LIN {X 0,Y 188.988,Z 308.592,A -85,B 0,C 180,E1 -22467.201,E2 -22467.201} C_VEL
LIN {X 0,Y 185.39,Z 303.655,A -85,B 0,C 180,E1 -22469.376,E2 -22469.376} C_VEL
LIN {X 0,Y 183.716,Z 298.969,A -85,B 0,C 180,E1 -22473.901,E2 -22473.901} C_VEL
LIN {X 0,Y 182.459,Z 295.961,A -85,B 0,C 180,E1 -22477.581,E2 -22477.581} C_VEL
LIN {X 0,Y 181.404,Z 292.928,A -85,B 0,C 180,E1 -22481.945,E2 -22481.945} C_VEL
LIN {X 0,Y 180.335,Z 289.551,A -85,B 0,C 180,E1 -22488.764,E2 -22488.764} C_VEL
LIN {X 0,Y 179.767,Z 288.375,A -85,B 0,C 180,E1 -22493.265,E2 -22493.265} C_VEL
LIN {X 0,Y 179.829,Z 287.586,A -85,B 0,C 180,E1 -22500.001,E2 -22500.001} C_VEL
LIN {X 0,Y 180.049,Z 288.87,A -85,B 0,C 180,E1 -22507.094,E2 -22507.094} C_VEL
LIN {X 0,Y 180.404,Z 289.347,A -85,B 0,C 180,E1 -22508.966,E2 -22508.966} C_VEL
LIN {X 0,Y 181.337,Z 292.707,A -85,B 0,C 180,E1 -22515.742,E2 -22515.742} C_VEL
LIN {X 0,Y 182.454,Z 295.747,A -85,B 0,C 180,E1 -22520.285,E2 -22520.285} C_VEL
LIN {X 0,Y 183.828,Z 299.51,A -85,B 0,C 180,E1 -22524.87,E2 -22524.87} C_VEL
LIN {X 0,Y 185.464,Z 304.104,A -85,B 0,C 180,E1 -22529.514,E2 -22529.514} C_VEL
LIN {X 0,Y 186.625,Z 307.65,A -85,B 0,C 180,E1 -22532.354,E2 -22532.354} C_VEL
LIN {X 0,Y 190.377,Z 313.038,A -85,B 0,C 180,E1 -22534.503,E2 -22534.503} C_VEL
LIN {X 0,Y 194.923,Z 320.088,A -85,B 0,C 180,E1 -22536.853,E2 -22536.853} C_VEL
LIN {X 0,Y 200.843,Z 329.671,A -85,B 0,C 180,E1 -22539.608,E2 -22539.608} C_VEL
LIN {X 0,Y 207.054,Z 341.003,A -85,B 0,C 180,E1 -22542.242,E2 -22542.242} C_VEL
LIN {X 0,Y 213.308,Z 354.054,A -85,B 0,C 180,E1 -22544.675,E2 -22544.675} C_VEL
LIN {X 0,Y 215.63,Z 359.84,A -85,B 0,C 180,E1 -22545.558,E2 -22545.558} C_VEL
LIN {X 0,Y 216.978,Z 371.187,A -85,B 0,C 180,E1 -22546.403,E2 -22546.403} C_VEL
LIN {X 0,Y 213.581,Z 427.914,A -85,B 0,C 180,E1 -22548.075,E2 -22548.075} C_VEL
LIN {X 0,Y 211.9,Z 441.326,A -85,B 0,C 180,E1 -22548.763,E2 -22548.763} C_VEL
LIN {X 0,Y 209.528,Z 454.408,A -85,B 0,C 180,E1 -22549.784,E2 -22549.784} C_VEL
LIN {X 0,Y 206.842,Z 466.094,A -85,B 0,C 180,E1 -22551.055,E2 -22551.055} C_VEL
LIN {X 0,Y 203.672,Z 477.504,A -85,B 0,C 180,E1 -22552.686,E2 -22552.686} C_VEL
LIN {X 0,Y 200.113,Z 487.996,A -85,B 0,C 180,E1 -22554.586,E2 -22554.586} C_VEL
LIN {X 0,Y 196.107,Z 497.993,A -85,B 0,C 180,E1 -22556.872,E2 -22556.872} C_VEL
LIN {X 0,Y 192.484,Z 506.265,A -85,B 0,C 180,E1 -22559.259,E2 -22559.259} C_VEL
LIN {X 0,Y 188.562,Z 514.429,A -85,B 0,C 180,E1 -22562.232,E2 -22562.232} C_VEL
LIN {X 0,Y 185.25,Z 521.075,A -85,B 0,C 180,E1 -22565.335,E2 -22565.335} C_VEL
LIN {X 0,Y 182.489,Z 526.45,A -85,B 0,C 180,E1 -22568.54,E2 -22568.54} C_VEL
LIN {X 0,Y 180.226,Z 530.729,A -85,B 0,C 180,E1 -22571.823,E2 -22571.823} C_VEL
LIN {X 0,Y 178.925,Z 533.018,A -85,B 0,C 180,E1 -22574.041,E2 -22574.041} C_VEL
LIN {X 0,Y 177.241,Z 536.394,A -85,B 0,C 180,E1 -22578.565,E2 -22578.565} C_VEL
LIN {X 0,Y 176.7,Z 537.498,A -85,B 0,C 180,E1 -22580.846,E2 -22580.846} C_VEL
LIN {X 0,Y 176.115,Z 538.572,A -85,B 0,C 180,E1 -22585.422,E2 -22585.422} C_VEL
LIN {X 0,Y 176.114,Z 538.233,A -85,B 0,C 180,E1 -22590,E2 -22590} C_VEL
LIN {X 0,Y 176.586,Z 536.474,A -85,B 0,C 180,E1 -22594.565,E2 -22594.565} C_VEL
LIN {X 0,Y 177.693,Z 533.161,A -85,B 0,C 180,E1 -22599.102,E2 -22599.102} C_VEL
LIN {X 0,Y 179.055,Z 529.638,A -85,B 0,C 180,E1 -22602.467,E2 -22602.467} C_VEL
LIN {X 0,Y 180.92,Z 525.106,A -85,B 0,C 180,E1 -22605.778,E2 -22605.778} C_VEL
LIN {X 0,Y 183.79,Z 518.335,A -85,B 0,C 180,E1 -22609.547,E2 -22609.547} C_VEL
LIN {X 0,Y 186.845,Z 511.095,A -85,B 0,C 180,E1 -22612.677,E2 -22612.677} C_VEL
LIN {X 0,Y 190.293,Z 502.209,A -85,B 0,C 180,E1 -22615.718,E2 -22615.718} C_VEL
LIN {X 0,Y 193.973,Z 492.174,A -85,B 0,C 180,E1 -22618.394,E2 -22618.394} C_VEL
LIN {X 0,Y 197.187,Z 482.065,A -85,B 0,C 180,E1 -22620.522,E2 -22620.522} C_VEL
LIN {X 0,Y 200.625,Z 469.958,A -85,B 0,C 180,E1 -22622.485,E2 -22622.485} C_VEL
LIN {X 0,Y 203.442,Z 457.934,A -85,B 0,C 180,E1 -22623.971,E2 -22623.971} C_VEL
LIN {X 0,Y 205.741,Z 444.65,A -85,B 0,C 180,E1 -22625.199,E2 -22625.199} C_VEL
LIN {X 0,Y 207.478,Z 431.116,A -85,B 0,C 180,E1 -22626.008,E2 -22626.008} C_VEL
LIN {X 0,Y 208.695,Z 413.538,A -85,B 0,C 180,E1 -22626.617,E2 -22626.617} C_VEL
LIN {X 0,Y 211.032,Z 367.372,A -85,B 0,C 180,E1 -22628.031,E2 -22628.031} C_VEL
LIN {X 0,Y 209.082,Z 351.343,A -85,B 0,C 180,E1 -22629.173,E2 -22629.173} C_VEL
LIN {X 0,Y 202.802,Z 337.342,A -85,B 0,C 180,E1 -22631.415,E2 -22631.415} C_VEL
LIN {X 0,Y 197.38,Z 326.733,A -85,B 0,C 180,E1 -22633.468,E2 -22633.468} C_VEL
LIN {X 0,Y 191.774,Z 317.194,A -85,B 0,C 180,E1 -22635.727,E2 -22635.727} C_VEL
LIN {X 0,Y 188.452,Z 311.954,A -85,B 0,C 180,E1 -22637.158,E2 -22637.158} C_VEL
LIN {X 0,Y 185.851,Z 307.521,A -85,B 0,C 180,E1 -22638.52,E2 -22638.52} C_VEL
LIN {X 0,Y 184.237,Z 302.058,A -85,B 0,C 180,E1 -22642.385,E2 -22642.385} C_VEL
LIN {X 0,Y 182.761,Z 297.513,A -85,B 0,C 180,E1 -22646.11,E2 -22646.11} C_VEL
LIN {X 0,Y 180.979,Z 292.372,A -85,B 0,C 180,E1 -22650.959,E2 -22650.959} C_VEL
LIN {X 0,Y 179.769,Z 289.141,A -85,B 0,C 180,E1 -22654.529,E2 -22654.529} C_VEL
LIN {X 0,Y 178.544,Z 285.92,A -85,B 0,C 180,E1 -22658.949,E2 -22658.949} C_VEL
LIN {X 0,Y 178.648,Z 285.846,A -85,B 0,C 180,E1 -22661.655,E2 -22661.655} C_VEL
LIN {X 0,Y 178.655,Z 285.843,A -85,B 0,C 180,E1 -22666.347,E2 -22666.347} C_VEL
LIN {X 0,Y 178.912,Z 285.807,A -85,B 0,C 180,E1 -22670.959,E2 -22670.959} C_VEL
LIN {X 0,Y 178.864,Z 285.81,A -85,B 0,C 180,E1 -22675.492,E2 -22675.492} C_VEL
LIN {X 0,Y 179.367,Z 285.749,A -85,B 0,C 180,E1 -22679.999,E2 -22679.999} C_VEL
LIN {X 0,Y 178.869,Z 285.817,A -85,B 0,C 180,E1 -22684.506,E2 -22684.506} C_VEL
LIN {X 0,Y 178.935,Z 285.816,A -85,B 0,C 180,E1 -22689.038,E2 -22689.038} C_VEL
LIN {X 0,Y 178.657,Z 285.857,A -85,B 0,C 180,E1 -22693.652,E2 -22693.652} C_VEL
LIN {X 0,Y 178.623,Z 286.004,A -85,B 0,C 180,E1 -22699.327,E2 -22699.327} C_VEL
LIN {X 0,Y 179.991,Z 289.783,A -85,B 0,C 180,E1 -22704.203,E2 -22704.203} C_VEL
LIN {X 0,Y 181.21,Z 293.097,A -85,B 0,C 180,E1 -22707.736,E2 -22707.736} C_VEL
LIN {X 0,Y 183.125,Z 298.362,A -85,B 0,C 180,E1 -22712.499,E2 -22712.499} C_VEL
LIN {X 0,Y 184.812,Z 303.336,A -85,B 0,C 180,E1 -22716.197,E2 -22716.197} C_VEL
LIN {X 0,Y 189.323,Z 310.216,A -85,B 0,C 180,E1 -22718.361,E2 -22718.361} C_VEL
LIN {X 0,Y 194.564,Z 318.216,A -85,B 0,C 180,E1 -22720.555,E2 -22720.555} C_VEL
LIN {X 0,Y 201.427,Z 330.245,A -85,B 0,C 180,E1 -22723.214,E2 -22723.214} C_VEL
LIN {X 0,Y 207.772,Z 343.107,A -85,B 0,C 180,E1 -22725.515,E2 -22725.515} C_VEL
LIN {X 0,Y 212.209,Z 353.469,A -85,B 0,C 180,E1 -22727.065,E2 -22727.065} C_VEL
LIN {X 0,Y 208.951,Z 409.204,A -85,B 0,C 180,E1 -22728.827,E2 -22728.827} C_VEL
LIN {X 0,Y 208.047,Z 415.053,A -85,B 0,C 180,E1 -22728.881,E2 -22728.881} C_VEL
LIN {X 0,Y 202.147,Z 433.973,A -85,B 0,C 180,E1 -22728.563,E2 -22728.563} C_VEL
LIN {X 0,Y 201.311,Z 437.801,A -85,B 0,C 180,E1 -22728.678,E2 -22728.678} C_VEL
LIN {X 0,Y 201.054,Z 439.716,A -85,B 0,C 180,E1 -22728.791,E2 -22728.791} C_VEL
LIN {X 0,Y 198.753,Z 453.725,A -85,B 0,C 180,E1 -22729.811,E2 -22729.811} C_VEL
LIN {X 0,Y 196.069,Z 466.519,A -85,B 0,C 180,E1 -22731.151,E2 -22731.151} C_VEL
LIN {X 0,Y 192.593,Z 479.599,A -85,B 0,C 180,E1 -22732.98,E2 -22732.98} C_VEL
LIN {X 0,Y 188.999,Z 491.567,A -85,B 0,C 180,E1 -22735.187,E2 -22735.187} C_VEL
LIN {X 0,Y 185.68,Z 501.033,A -85,B 0,C 180,E1 -22737.361,E2 -22737.361} C_VEL
LIN {X 0,Y 181.482,Z 511.683,A -85,B 0,C 180,E1 -22740.413,E2 -22740.413} C_VEL
LIN {X 0,Y 178.053,Z 520.388,A -85,B 0,C 180,E1 -22743.638,E2 -22743.638} C_VEL
LIN {X 0,Y 174.916,Z 528.205,A -85,B 0,C 180,E1 -22747.332,E2 -22747.332} C_VEL
LIN {X 0,Y 172.603,Z 534.285,A -85,B 0,C 180,E1 -22750.99,E2 -22750.99} C_VEL
LIN {X 0,Y 170.858,Z 538.9,A -85,B 0,C 180,E1 -22754.493,E2 -22754.493} C_VEL
LIN {X 0,Y 169.722,Z 542.492,A -85,B 0,C 180,E1 -22758.051,E2 -22758.051} C_VEL
LIN {X 0,Y 169.28,Z 544.407,A -85,B 0,C 180,E1 -22760.441,E2 -22760.441} C_VEL
LIN {X 0,Y 168.849,Z 547.061,A -85,B 0,C 180,E1 -22765.225,E2 -22765.225} C_VEL
LIN {X 0,Y 168.983,Z 548.218,A -85,B 0,C 180,E1 -22770,E2 -22770} C_VEL
LIN {X 0,Y 168.89,Z 548.208,A -85,B 0,C 180,E1 -22772.921,E2 -22772.921} C_VEL
LIN {X 0,Y 168.991,Z 547.226,A -85,B 0,C 180,E1 -22777.167,E2 -22777.167} C_VEL
LIN {X 0,Y 169.78,Z 544.762,A -85,B 0,C 180,E1 -22781.945,E2 -22781.945} C_VEL
LIN {X 0,Y 170.968,Z 541.886,A -85,B 0,C 180,E1 -22785.497,E2 -22785.497} C_VEL
LIN {X 0,Y 173.498,Z 536.673,A -85,B 0,C 180,E1 -22790.14,E2 -22790.14} C_VEL
LIN {X 0,Y 175.919,Z 531.55,A -85,B 0,C 180,E1 -22793.547,E2 -22793.547} C_VEL
LIN {X 0,Y 179.575,Z 524.164,A -85,B 0,C 180,E1 -22797.378,E2 -22797.378} C_VEL
LIN {X 0,Y 183.322,Z 516.339,A -85,B 0,C 180,E1 -22800.528,E2 -22800.528} C_VEL
LIN {X 0,Y 187.683,Z 506.803,A -85,B 0,C 180,E1 -22803.526,E2 -22803.526} C_VEL
LIN {X 0,Y 191.637,Z 497.209,A -85,B 0,C 180,E1 -22805.928,E2 -22805.928} C_VEL
LIN {X 0,Y 195.407,Z 486.819,A -85,B 0,C 180,E1 -22808.018,E2 -22808.018} C_VEL
LIN {X 0,Y 199.458,Z 473.997,A -85,B 0,C 180,E1 -22810.019,E2 -22810.019} C_VEL
LIN {X 0,Y 202.815,Z 461.325,A -85,B 0,C 180,E1 -22811.507,E2 -22811.507} C_VEL
LIN {X 0,Y 205.587,Z 448.261,A -85,B 0,C 180,E1 -22812.632,E2 -22812.632} C_VEL
LIN {X 0,Y 207.681,Z 434.633,A -85,B 0,C 180,E1 -22813.435,E2 -22813.435} C_VEL
LIN {X 0,Y 209.176,Z 417.644,A -85,B 0,C 180,E1 -22814.044,E2 -22814.044} C_VEL
LIN {X 0,Y 212.691,Z 361.582,A -85,B 0,C 180,E1 -22815.805,E2 -22815.805} C_VEL
LIN {X 0,Y 206.911,Z 348.829,A -85,B 0,C 180,E1 -22818.115,E2 -22818.115} C_VEL
LIN {X 0,Y 201.177,Z 337.852,A -85,B 0,C 180,E1 -22820.553,E2 -22820.553} C_VEL
LIN {X 0,Y 195.155,Z 327.838,A -85,B 0,C 180,E1 -22823.331,E2 -22823.331} C_VEL
LIN {X 0,Y 189.772,Z 319.519,A -85,B 0,C 180,E1 -22826.095,E2 -22826.095} C_VEL
LIN {X 0,Y 186.099,Z 314.359,A -85,B 0,C 180,E1 -22828.162,E2 -22828.162} C_VEL
LIN {X 0,Y 181.851,Z 308.686,A -85,B 0,C 180,E1 -22830.802,E2 -22830.802} C_VEL
LIN {X 0,Y 178.233,Z 303.751,A -85,B 0,C 180,E1 -22833.509,E2 -22833.509} C_VEL
LIN {X 0,Y 176.472,Z 299.364,A -85,B 0,C 180,E1 -22838.997,E2 -22838.997} C_VEL
LIN {X 0,Y 175.428,Z 296.432,A -85,B 0,C 180,E1 -22843.715,E2 -22843.715} C_VEL
LIN {X 0,Y 174.827,Z 294.233,A -85,B 0,C 180,E1 -22848.405,E2 -22848.405} C_VEL
LIN {X 0,Y 174.62,Z 293.43,A -85,B 0,C 180,E1 -22850.736,E2 -22850.736} C_VEL
LIN {X 0,Y 174.209,Z 292.288,A -85,B 0,C 180,E1 -22857.689,E2 -22857.689} C_VEL
LIN {X 0,Y 174.368,Z 292.137,A -85,B 0,C 180,E1 -22860.001,E2 -22860.001} C_VEL
LIN {X 0,Y 174.572,Z 293.41,A -85,B 0,C 180,E1 -22867.151,E2 -22867.151} C_VEL
LIN {X 0,Y 174.898,Z 293.994,A -85,B 0,C 180,E1 -22869.25,E2 -22869.25} C_VEL
LIN {X 0,Y 175.921,Z 297.612,A -85,B 0,C 180,E1 -22876.508,E2 -22876.508} C_VEL
LIN {X 0,Y 176.956,Z 300.581,A -85,B 0,C 180,E1 -22880.944,E2 -22880.944} C_VEL
LIN {X 0,Y 178.332,Z 304.501,A -85,B 0,C 180,E1 -22885.691,E2 -22885.691} C_VEL
LIN {X 0,Y 179.408,Z 307.362,A -85,B 0,C 180,E1 -22888.426,E2 -22888.426} C_VEL
LIN {X 0,Y 183.53,Z 313.038,A -85,B 0,C 180,E1 -22891.21,E2 -22891.21} C_VEL
LIN {X 0,Y 188.311,Z 320.152,A -85,B 0,C 180,E1 -22894.044,E2 -22894.044} C_VEL
LIN {X 0,Y 191.838,Z 325.708,A -85,B 0,C 180,E1 -22895.943,E2 -22895.943} C_VEL
LIN {X 0,Y 197.44,Z 335.085,A -85,B 0,C 180,E1 -22898.694,E2 -22898.694} C_VEL
LIN {X 0,Y 203.749,Z 346.971,A -85,B 0,C 180,E1 -22901.501,E2 -22901.501} C_VEL
LIN {X 0,Y 209.488,Z 359.433,A -85,B 0,C 180,E1 -22903.85,E2 -22903.85} C_VEL
LIN {X 0,Y 210.867,Z 363.303,A -85,B 0,C 180,E1 -22904.421,E2 -22904.421} C_VEL
LIN {X 0,Y 211.836,Z 372.835,A -85,B 0,C 180,E1 -22905.125,E2 -22905.125} C_VEL
LIN {X 0,Y 208.375,Z 427.933,A -85,B 0,C 180,E1 -22906.767,E2 -22906.767} C_VEL
LIN {X 0,Y 206.627,Z 441.435,A -85,B 0,C 180,E1 -22907.468,E2 -22907.468} C_VEL
LIN {X 0,Y 204.15,Z 454.506,A -85,B 0,C 180,E1 -22908.495,E2 -22908.495} C_VEL
LIN {X 0,Y 201.385,Z 466.19,A -85,B 0,C 180,E1 -22909.789,E2 -22909.789} C_VEL
LIN {X 0,Y 198.045,Z 477.602,A -85,B 0,C 180,E1 -22911.435,E2 -22911.435} C_VEL
LIN {X 0,Y 194.365,Z 488.1,A -85,B 0,C 180,E1 -22913.372,E2 -22913.372} C_VEL
LIN {X 0,Y 190.195,Z 498.105,A -85,B 0,C 180,E1 -22915.702,E2 -22915.702} C_VEL
LIN {X 0,Y 186.413,Z 506.385,A -85,B 0,C 180,E1 -22918.142,E2 -22918.142} C_VEL
LIN {X 0,Y 182.303,Z 514.558,A -85,B 0,C 180,E1 -22921.192,E2 -22921.192} C_VEL
LIN {X 0,Y 178.787,Z 521.213,A -85,B 0,C 180,E1 -22924.38,E2 -22924.38} C_VEL
LIN {X 0,Y 175.863,Z 526.599,A -85,B 0,C 180,E1 -22927.689,E2 -22927.689} C_VEL
LIN {X 0,Y 173.47,Z 530.888,A -85,B 0,C 180,E1 -22931.088,E2 -22931.088} C_VEL
LIN {X 0,Y 172.075,Z 533.182,A -85,B 0,C 180,E1 -22933.388,E2 -22933.388} C_VEL
LIN {X 0,Y 170.27,Z 536.568,A -85,B 0,C 180,E1 -22938.09,E2 -22938.09} C_VEL
LIN {X 0,Y 169.674,Z 537.682,A -85,B 0,C 180,E1 -22940.463,E2 -22940.463} C_VEL
LIN {X 0,Y 169.028,Z 538.768,A -85,B 0,C 180,E1 -22945.23,E2 -22945.23} C_VEL
LIN {X 0,Y 169.024,Z 538.441,A -85,B 0,C 180,E1 -22950,E2 -22950} C_VEL
LIN {X 0,Y 169.52,Z 536.696,A -85,B 0,C 180,E1 -22954.756,E2 -22954.756} C_VEL
LIN {X 0,Y 170.691,Z 533.4,A -85,B 0,C 180,E1 -22959.479,E2 -22959.479} C_VEL
LIN {X 0,Y 172.727,Z 528.497,A -85,B 0,C 180,E1 -22964.13,E2 -22964.13} C_VEL
LIN {X 0,Y 174.915,Z 523.6,A -85,B 0,C 180,E1 -22967.538,E2 -22967.538} C_VEL
LIN {X 0,Y 178.166,Z 516.415,A -85,B 0,C 180,E1 -22971.4,E2 -22971.4} C_VEL
LIN {X 0,Y 181.505,Z 508.678,A -85,B 0,C 180,E1 -22974.597,E2 -22974.597} C_VEL
LIN {X 0,Y 185.368,Z 499.143,A -85,B 0,C 180,E1 -22977.674,E2 -22977.674} C_VEL
LIN {X 0,Y 188.94,Z 489.408,A -85,B 0,C 180,E1 -22980.142,E2 -22980.142} C_VEL
LIN {X 0,Y 192.342,Z 478.69,A -85,B 0,C 180,E1 -22982.301,E2 -22982.301} C_VEL
LIN {X 0,Y 195.657,Z 467.131,A -85,B 0,C 180,E1 -22984.071,E2 -22984.071} C_VEL
LIN {X 0,Y 198.523,Z 454.168,A -85,B 0,C 180,E1 -22985.583,E2 -22985.583} C_VEL
LIN {X 0,Y 200.692,Z 441.123,A -85,B 0,C 180,E1 -22986.683,E2 -22986.683} C_VEL
LIN {X 0,Y 202.257,Z 428.164,A -85,B 0,C 180,E1 -22987.39,E2 -22987.39} C_VEL
LIN {X 0,Y 205.638,Z 368.57,A -85,B 0,C 180,E1 -22989.267,E2 -22989.267} C_VEL
LIN {X 0,Y 203.986,Z 354.351,A -85,B 0,C 180,E1 -22990.318,E2 -22990.318} C_VEL
LIN {X 0,Y 198.265,Z 341.326,A -85,B 0,C 180,E1 -22992.492,E2 -22992.492} C_VEL
LIN {X 0,Y 193.104,Z 331.102,A -85,B 0,C 180,E1 -22994.565,E2 -22994.565} C_VEL
LIN {X 0,Y 187.912,Z 322.048,A -85,B 0,C 180,E1 -22996.788,E2 -22996.788} C_VEL
LIN {X 0,Y 184.709,Z 316.898,A -85,B 0,C 180,E1 -22998.25,E2 -22998.25} C_VEL
LIN {X 0,Y 181.35,Z 311.778,A -85,B 0,C 180,E1 -22999.876,E2 -22999.876} C_VEL
LIN {X 0,Y 178.713,Z 307.363,A -85,B 0,C 180,E1 -23001.418,E2 -23001.418} C_VEL
LIN {X 0,Y 177.335,Z 302.898,A -85,B 0,C 180,E1 -23004.924,E2 -23004.924} C_VEL
LIN {X 0,Y 175.96,Z 298.779,A -85,B 0,C 180,E1 -23008.718,E2 -23008.718} C_VEL
LIN {X 0,Y 174.787,Z 295.473,A -85,B 0,C 180,E1 -23012.2,E2 -23012.2} C_VEL
LIN {X 0,Y 172.929,Z 290.476,A -85,B 0,C 180,E1 -23018.544,E2 -23018.544} C_VEL
LIN {X 0,Y 171.589,Z 286.754,A -85,B 0,C 180,E1 -23025.47,E2 -23025.47} C_VEL
LIN {X 0,Y 171.848,Z 286.685,A -85,B 0,C 180,E1 -23030.584,E2 -23030.584} C_VEL
LIN {X 0,Y 171.813,Z 286.688,A -85,B 0,C 180,E1 -23035.307,E2 -23035.307} C_VEL
LIN {X 0,Y 172.329,Z 286.625,A -85,B 0,C 180,E1 -23039.999,E2 -23039.999} C_VEL
LIN {X 0,Y 171.818,Z 286.693,A -85,B 0,C 180,E1 -23044.692,E2 -23044.692} C_VEL
LIN {X 0,Y 171.87,Z 286.691,A -85,B 0,C 180,E1 -23049.413,E2 -23049.413} C_VEL
LIN {X 0,Y 171.647,Z 286.964,A -85,B 0,C 180,E1 -23053.315,E2 -23053.315} C_VEL
LIN {X 0,Y 172.896,Z 290.092,A -85,B 0,C 180,E1 -23058.976,E2 -23058.976} C_VEL
LIN {X 0,Y 174.536,Z 294.799,A -85,B 0,C 180,E1 -23065.011,E2 -23065.011} C_VEL
LIN {X 0,Y 176.266,Z 299.567,A -85,B 0,C 180,E1 -23069.893,E2 -23069.893} C_VEL
LIN {X 0,Y 177.686,Z 303.491,A -85,B 0,C 180,E1 -23073.206,E2 -23073.206} C_VEL
LIN {X 0,Y 181.057,Z 308.371,A -85,B 0,C 180,E1 -23075.097,E2 -23075.097} C_VEL
LIN {X 0,Y 185.961,Z 315.797,A -85,B 0,C 180,E1 -23077.474,E2 -23077.474} C_VEL
LIN {X 0,Y 190.798,Z 323.362,A -85,B 0,C 180,E1 -23079.609,E2 -23079.609} C_VEL
LIN {X 0,Y 197.137,Z 334.68,A -85,B 0,C 180,E1 -23082.204,E2 -23082.204} C_VEL
LIN {X 0,Y 203.357,Z 347.627,A -85,B 0,C 180,E1 -23084.598,E2 -23084.598} C_VEL
LIN {X 0,Y 206.717,Z 355.627,A -85,B 0,C 180,E1 -23085.844,E2 -23085.844} C_VEL
LIN {X 0,Y 202.135,Z 429.954,A -85,B 0,C 180,E1 -23088.276,E2 -23088.276} C_VEL
LIN {X 0,Y 201.054,Z 439.716,A -85,B 0,C 180,E1 -23088.791,E2 -23088.791} C_VEL
LIN {X 0,Y 199.788,Z 445.41,A -85,B 0,C 180,E1 -23089.055,E2 -23089.055} C_VEL
LIN {X 0,Y 195.958,Z 454.527,A -85,B 0,C 180,E1 -23089.273,E2 -23089.273} C_VEL
LIN {X 0,Y 191.716,Z 463.419,A -85,B 0,C 180,E1 -23089.648,E2 -23089.648} C_VEL
LIN {X 0,Y 189.822,Z 468.738,A -85,B 0,C 180,E1 -23090.164,E2 -23090.164} C_VEL
LIN {X 0,Y 186.5,Z 480.541,A -85,B 0,C 180,E1 -23091.899,E2 -23091.899} C_VEL
LIN {X 0,Y 183.013,Z 491.653,A -85,B 0,C 180,E1 -23094.021,E2 -23094.021} C_VEL
LIN {X 0,Y 178.929,Z 502.623,A -85,B 0,C 180,E1 -23096.641,E2 -23096.641} C_VEL
LIN {X 0,Y 175.293,Z 511.339,A -85,B 0,C 180,E1 -23099.258,E2 -23099.258} C_VEL
LIN {X 0,Y 171.658,Z 520.079,A -85,B 0,C 180,E1 -23102.575,E2 -23102.575} C_VEL
LIN {X 0,Y 168.197,Z 528.201,A -85,B 0,C 180,E1 -23106.549,E2 -23106.549} C_VEL
LIN {X 0,Y 165.857,Z 534.023,A -85,B 0,C 180,E1 -23110.185,E2 -23110.185} C_VEL
LIN {X 0,Y 163.985,Z 538.65,A -85,B 0,C 180,E1 -23113.825,E2 -23113.825} C_VEL
LIN {X 0,Y 162.739,Z 542.253,A -85,B 0,C 180,E1 -23117.53,E2 -23117.53} C_VEL
LIN {X 0,Y 161.904,Z 545.708,A -85,B 0,C 180,E1 -23122.518,E2 -23122.518} C_VEL
LIN {X 0,Y 161.755,Z 547.613,A -85,B 0,C 180,E1 -23127.51,E2 -23127.51} C_VEL
LIN {X 0,Y 161.894,Z 548.017,A -85,B 0,C 180,E1 -23130,E2 -23130} C_VEL
LIN {X 0,Y 161.795,Z 548.051,A -85,B 0,C 180,E1 -23132.49,E2 -23132.49} C_VEL
LIN {X 0,Y 161.928,Z 547.04,A -85,B 0,C 180,E1 -23137.482,E2 -23137.482} C_VEL
LIN {X 0,Y 162.791,Z 544.584,A -85,B 0,C 180,E1 -23142.466,E2 -23142.466} C_VEL
LIN {X 0,Y 164.096,Z 541.719,A -85,B 0,C 180,E1 -23146.164,E2 -23146.164} C_VEL
LIN {X 0,Y 166.807,Z 536.515,A -85,B 0,C 180,E1 -23150.985,E2 -23150.985} C_VEL
LIN {X 0,Y 169.371,Z 531.4,A -85,B 0,C 180,E1 -23154.516,E2 -23154.516} C_VEL
LIN {X 0,Y 173.246,Z 524.024,A -85,B 0,C 180,E1 -23158.467,E2 -23158.467} C_VEL
LIN {X 0,Y 177.196,Z 516.207,A -85,B 0,C 180,E1 -23161.703,E2 -23161.703} C_VEL
LIN {X 0,Y 181.793,Z 506.678,A -85,B 0,C 180,E1 -23164.765,E2 -23164.765} C_VEL
LIN {X 0,Y 186.336,Z 496.031,A -85,B 0,C 180,E1 -23167.452,E2 -23167.452} C_VEL
LIN {X 0,Y 190.287,Z 485.405,A -85,B 0,C 180,E1 -23169.576,E2 -23169.576} C_VEL
LIN {X 0,Y 194.072,Z 473.879,A -85,B 0,C 180,E1 -23171.367,E2 -23171.367} C_VEL
LIN {X 0,Y 197.564,Z 461.203,A -85,B 0,C 180,E1 -23172.869,E2 -23172.869} C_VEL
LIN {X 0,Y 200.551,Z 447.38,A -85,B 0,C 180,E1 -23174.058,E2 -23174.058} C_VEL
LIN {X 0,Y 202.742,Z 433.134,A -85,B 0,C 180,E1 -23174.873,E2 -23174.873} C_VEL
LIN {X 0,Y 204.401,Z 413.511,A -85,B 0,C 180,E1 -23175.547,E2 -23175.547} C_VEL
LIN {X 0,Y 207.608,Z 363.936,A -85,B 0,C 180,E1 -23177.128,E2 -23177.128} C_VEL
LIN {X 0,Y 201.268,Z 350.06,A -85,B 0,C 180,E1 -23179.842,E2 -23179.842} C_VEL
LIN {X 0,Y 195.295,Z 338.908,A -85,B 0,C 180,E1 -23182.602,E2 -23182.602} C_VEL
LIN {X 0,Y 189.819,Z 329.842,A -85,B 0,C 180,E1 -23185.383,E2 -23185.383} C_VEL
LIN {X 0,Y 185.485,Z 323.326,A -85,B 0,C 180,E1 -23187.808,E2 -23187.808} C_VEL
LIN {X 0,Y 183.331,Z 320.171,A -85,B 0,C 180,E1 -23189.115,E2 -23189.115} C_VEL
LIN {X 0,Y 179.443,Z 314.792,A -85,B 0,C 180,E1 -23191.667,E2 -23191.667} C_VEL
LIN {X 0,Y 175.385,Z 309.519,A -85,B 0,C 180,E1 -23194.68,E2 -23194.68} C_VEL
LIN {X 0,Y 171.063,Z 304.168,A -85,B 0,C 180,E1 -23198.616,E2 -23198.616} C_VEL
LIN {X 0,Y 170.003,Z 301.235,A -85,B 0,C 180,E1 -23203.18,E2 -23203.18} C_VEL
LIN {X 0,Y 169.334,Z 298.913,A -85,B 0,C 180,E1 -23208.024,E2 -23208.024} C_VEL
LIN {X 0,Y 169.15,Z 298.05,A -85,B 0,C 180,E1 -23210.434,E2 -23210.434} C_VEL
LIN {X 0,Y 168.67,Z 297.177,A -85,B 0,C 180,E1 -23215.221,E2 -23215.221} C_VEL
LIN {X 0,Y 168.906,Z 296.688,A -85,B 0,C 180,E1 -23220.001,E2 -23220.001} C_VEL
LIN {X 0,Y 169.114,Z 297.927,A -85,B 0,C 180,E1 -23227.189,E2 -23227.189} C_VEL
LIN {X 0,Y 169.406,Z 298.635,A -85,B 0,C 180,E1 -23229.553,E2 -23229.553} C_VEL
LIN {X 0,Y 169.909,Z 300.873,A -85,B 0,C 180,E1 -23234.371,E2 -23234.371} C_VEL
LIN {X 0,Y 170.867,Z 303.708,A -85,B 0,C 180,E1 -23239.212,E2 -23239.212} C_VEL
LIN {X 0,Y 172.147,Z 307.05,A -85,B 0,C 180,E1 -23243.457,E2 -23243.457} C_VEL
LIN {X 0,Y 176.113,Z 312.387,A -85,B 0,C 180,E1 -23246.837,E2 -23246.837} C_VEL
LIN {X 0,Y 178.142,Z 315.199,A -85,B 0,C 180,E1 -23248.355,E2 -23248.355} C_VEL
LIN {X 0,Y 181.763,Z 320.287,A -85,B 0,C 180,E1 -23250.82,E2 -23250.82} C_VEL
LIN {X 0,Y 185.491,Z 325.949,A -85,B 0,C 180,E1 -23253.12,E2 -23253.12} C_VEL
LIN {X 0,Y 189.11,Z 331.89,A -85,B 0,C 180,E1 -23255.173,E2 -23255.173} C_VEL
LIN {X 0,Y 194.164,Z 340.57,A -85,B 0,C 180,E1 -23257.781,E2 -23257.781} C_VEL
LIN {X 0,Y 199.896,Z 351.759,A -85,B 0,C 180,E1 -23260.475,E2 -23260.475} C_VEL
LIN {X 0,Y 205.015,Z 363.097,A -85,B 0,C 180,E1 -23262.699,E2 -23262.699} C_VEL
LIN {X 0,Y 206.108,Z 365.908,A -85,B 0,C 180,E1 -23263.166,E2 -23263.166} C_VEL
LIN {X 0,Y 206.863,Z 373.468,A -85,B 0,C 180,E1 -23263.753,E2 -23263.753} C_VEL
LIN {X 0,Y 203.268,Z 428.067,A -85,B 0,C 180,E1 -23265.398,E2 -23265.398} C_VEL
LIN {X 0,Y 201.469,Z 441.545,A -85,B 0,C 180,E1 -23266.108,E2 -23266.108} C_VEL
LIN {X 0,Y 198.903,Z 454.604,A -85,B 0,C 180,E1 -23267.143,E2 -23267.143} C_VEL
LIN {X 0,Y 196.02,Z 466.285,A -85,B 0,C 180,E1 -23268.449,E2 -23268.449} C_VEL
LIN {X 0,Y 192.279,Z 478.472,A -85,B 0,C 180,E1 -23270.245,E2 -23270.245} C_VEL
LIN {X 0,Y 188.258,Z 489.272,A -85,B 0,C 180,E1 -23272.317,E2 -23272.317} C_VEL
LIN {X 0,Y 183.501,Z 499.986,A -85,B 0,C 180,E1 -23274.937,E2 -23274.937} C_VEL
LIN {X 0,Y 178.934,Z 509.446,A -85,B 0,C 180,E1 -23277.979,E2 -23277.979} C_VEL
LIN {X 0,Y 174.771,Z 517.09,A -85,B 0,C 180,E1 -23281.148,E2 -23281.148} C_VEL
LIN {X 0,Y 171.209,Z 523.443,A -85,B 0,C 180,E1 -23284.569,E2 -23284.569} C_VEL
LIN {X 0,Y 168.404,Z 528.322,A -85,B 0,C 180,E1 -23287.939,E2 -23287.939} C_VEL
LIN {X 0,Y 165.962,Z 532.266,A -85,B 0,C 180,E1 -23291.482,E2 -23291.482} C_VEL
LIN {X 0,Y 164.182,Z 535.238,A -85,B 0,C 180,E1 -23295.118,E2 -23295.118} C_VEL
LIN {X 0,Y 162.67,Z 537.865,A -85,B 0,C 180,E1 -23300.048,E2 -23300.048} C_VEL
LIN {X 0,Y 161.946,Z 538.964,A -85,B 0,C 180,E1 -23305.021,E2 -23305.021} C_VEL
LIN {X 0,Y 161.935,Z 538.648,A -85,B 0,C 180,E1 -23310,E2 -23310} C_VEL
LIN {X 0,Y 162.447,Z 536.918,A -85,B 0,C 180,E1 -23314.964,E2 -23314.964} C_VEL
LIN {X 0,Y 163.708,Z 533.639,A -85,B 0,C 180,E1 -23319.888,E2 -23319.888} C_VEL
LIN {X 0,Y 165.237,Z 530.148,A -85,B 0,C 180,E1 -23323.528,E2 -23323.528} C_VEL
LIN {X 0,Y 167.322,Z 525.647,A -85,B 0,C 180,E1 -23327.098,E2 -23327.098} C_VEL
LIN {X 0,Y 170.508,Z 518.922,A -85,B 0,C 180,E1 -23331.14,E2 -23331.14} C_VEL
LIN {X 0,Y 173.85,Z 511.732,A -85,B 0,C 180,E1 -23334.479,E2 -23334.479} C_VEL
LIN {X 0,Y 177.637,Z 502.908,A -85,B 0,C 180,E1 -23337.701,E2 -23337.701} C_VEL
LIN {X 0,Y 181.658,Z 492.973,A -85,B 0,C 180,E1 -23340.515,E2 -23340.515} C_VEL
LIN {X 0,Y 185.147,Z 483.001,A -85,B 0,C 180,E1 -23342.745,E2 -23342.745} C_VEL
LIN {X 0,Y 188.728,Z 471.537,A -85,B 0,C 180,E1 -23344.717,E2 -23344.717} C_VEL
LIN {X 0,Y 191.7,Z 460.075,A -85,B 0,C 180,E1 -23346.238,E2 -23346.238} C_VEL
LIN {X 0,Y 194.162,Z 447.719,A -85,B 0,C 180,E1 -23347.484,E2 -23347.484} C_VEL
LIN {X 0,Y 196.24,Z 433.883,A -85,B 0,C 180,E1 -23348.435,E2 -23348.435} C_VEL
LIN {X 0,Y 197.456,Z 419.765,A -85,B 0,C 180,E1 -23349.012,E2 -23349.012} C_VEL
LIN {X 0,Y 200.365,Z 369.705,A -85,B 0,C 180,E1 -23350.567,E2 -23350.567} C_VEL
LIN {X 0,Y 198.883,Z 356.983,A -85,B 0,C 180,E1 -23351.565,E2 -23351.565} C_VEL
LIN {X 0,Y 192.971,Z 343.441,A -85,B 0,C 180,E1 -23353.972,E2 -23353.972} C_VEL
LIN {X 0,Y 187.433,Z 332.605,A -85,B 0,C 180,E1 -23356.372,E2 -23356.372} C_VEL
LIN {X 0,Y 181.632,Z 322.707,A -85,B 0,C 180,E1 -23359.097,E2 -23359.097} C_VEL
LIN {X 0,Y 178.164,Z 317.338,A -85,B 0,C 180,E1 -23360.864,E2 -23360.864} C_VEL
LIN {X 0,Y 174.821,Z 312.213,A -85,B 0,C 180,E1 -23362.705,E2 -23362.705} C_VEL
LIN {X 0,Y 171.559,Z 307.159,A -85,B 0,C 180,E1 -23364.824,E2 -23364.824} C_VEL
LIN {X 0,Y 170.08,Z 302.721,A -85,B 0,C 180,E1 -23368.9,E2 -23368.9} C_VEL
LIN {X 0,Y 168.866,Z 299.22,A -85,B 0,C 180,E1 -23372.753,E2 -23372.753} C_VEL
LIN {X 0,Y 167.442,Z 295.397,A -85,B 0,C 180,E1 -23377.804,E2 -23377.804} C_VEL
LIN {X 0,Y 166.287,Z 292.436,A -85,B 0,C 180,E1 -23382.791,E2 -23382.791} C_VEL
LIN {X 0,Y 165.962,Z 291.146,A -85,B 0,C 180,E1 -23385.28,E2 -23385.28} C_VEL
LIN {X 0,Y 165.274,Z 289.396,A -85,B 0,C 180,E1 -23390.206,E2 -23390.206} C_VEL
LIN {X 0,Y 164.923,Z 288.388,A -85,B 0,C 180,E1 -23395.11,E2 -23395.11} C_VEL
LIN {X 0,Y 165.325,Z 287.802,A -85,B 0,C 180,E1 -23399.999,E2 -23399.999} C_VEL
LIN {X 0,Y 165.022,Z 288.719,A -85,B 0,C 180,E1 -23404.885,E2 -23404.885} C_VEL
LIN {X 0,Y 165.565,Z 289.974,A -85,B 0,C 180,E1 -23409.775,E2 -23409.775} C_VEL
LIN {X 0,Y 166.079,Z 291.384,A -85,B 0,C 180,E1 -23413.276,E2 -23413.276} C_VEL
LIN {X 0,Y 167.362,Z 294.972,A -85,B 0,C 180,E1 -23419.629,E2 -23419.629} C_VEL
LIN {X 0,Y 168.741,Z 298.768,A -85,B 0,C 180,E1 -23424.613,E2 -23424.613} C_VEL
LIN {X 0,Y 170.318,Z 303.224,A -85,B 0,C 180,E1 -23429.331,E2 -23429.331} C_VEL
LIN {X 0,Y 171.217,Z 304.942,A -85,B 0,C 180,E1 -23430.272,E2 -23430.272} C_VEL
LIN {X 0,Y 175.383,Z 310.479,A -85,B 0,C 180,E1 -23432.749,E2 -23432.749} C_VEL
LIN {X 0,Y 179.262,Z 316.121,A -85,B 0,C 180,E1 -23434.849,E2 -23434.849} C_VEL
LIN {X 0,Y 182.774,Z 321.55,A -85,B 0,C 180,E1 -23436.614,E2 -23436.614} C_VEL
LIN {X 0,Y 187.362,Z 329.022,A -85,B 0,C 180,E1 -23438.751,E2 -23438.751} C_VEL
LIN {X 0,Y 193.082,Z 339.482,A -85,B 0,C 180,E1 -23441.225,E2 -23441.225} C_VEL
LIN {X 0,Y 198.88,Z 351.822,A -85,B 0,C 180,E1 -23443.59,E2 -23443.59} C_VEL
LIN {X 0,Y 201.328,Z 357.785,A -85,B 0,C 180,E1 -23444.559,E2 -23444.559} C_VEL
LIN {X 0,Y 196.654,Z 430.659,A -85,B 0,C 180,E1 -23446.998,E2 -23446.998} C_VEL
LIN {X 0,Y 194.869,Z 444.575,A -85,B 0,C 180,E1 -23447.802,E2 -23447.802} C_VEL
LIN {X 0,Y 192.404,Z 457.613,A -85,B 0,C 180,E1 -23448.892,E2 -23448.892} C_VEL
LIN {X 0,Y 189.822,Z 468.738,A -85,B 0,C 180,E1 -23450.164,E2 -23450.164} C_VEL
LIN {X 0,Y 187.879,Z 474.002,A -85,B 0,C 180,E1 -23450.755,E2 -23450.755} C_VEL
LIN {X 0,Y 183.175,Z 482.297,A -85,B 0,C 180,E1 -23451.565,E2 -23451.565} C_VEL
LIN {X 0,Y 178.206,Z 490.252,A -85,B 0,C 180,E1 -23452.573,E2 -23452.573} C_VEL
LIN {X 0,Y 175.885,Z 494.903,A -85,B 0,C 180,E1 -23453.48,E2 -23453.48} C_VEL
LIN {X 0,Y 171.433,Z 505.911,A -85,B 0,C 180,E1 -23456.397,E2 -23456.397} C_VEL
LIN {X 0,Y 167.221,Z 515.599,A -85,B 0,C 180,E1 -23459.713,E2 -23459.713} C_VEL
LIN {X 0,Y 163.613,Z 523.544,A -85,B 0,C 180,E1 -23463.191,E2 -23463.191} C_VEL
LIN {X 0,Y 160.695,Z 530.075,A -85,B 0,C 180,E1 -23466.821,E2 -23466.821} C_VEL
LIN {X 0,Y 158.428,Z 535.409,A -85,B 0,C 180,E1 -23470.567,E2 -23470.567} C_VEL
LIN {X 0,Y 156.555,Z 539.686,A -85,B 0,C 180,E1 -23474.375,E2 -23474.375} C_VEL
LIN {X 0,Y 155.203,Z 543.943,A -85,B 0,C 180,E1 -23479.565,E2 -23479.565} C_VEL
LIN {X 0,Y 154.842,Z 545.485,A -85,B 0,C 180,E1 -23482.174,E2 -23482.174} C_VEL
LIN {X 0,Y 154.678,Z 546.635,A -85,B 0,C 180,E1 -23484.786,E2 -23484.786} C_VEL
LIN {X 0,Y 154.792,Z 547.815,A -85,B 0,C 180,E1 -23490,E2 -23490} C_VEL
LIN {X 0,Y 154.696,Z 547.854,A -85,B 0,C 180,E1 -23492.604,E2 -23492.604} C_VEL
LIN {X 0,Y 154.861,Z 546.853,A -85,B 0,C 180,E1 -23497.825,E2 -23497.825} C_VEL
LIN {X 0,Y 155.826,Z 544.408,A -85,B 0,C 180,E1 -23503.033,E2 -23503.033} C_VEL
LIN {X 0,Y 157.251,Z 541.551,A -85,B 0,C 180,E1 -23506.888,E2 -23506.888} C_VEL
LIN {X 0,Y 160.151,Z 536.357,A -85,B 0,C 180,E1 -23511.901,E2 -23511.901} C_VEL
LIN {X 0,Y 162.885,Z 531.251,A -85,B 0,C 180,E1 -23515.56,E2 -23515.56} C_VEL
LIN {X 0,Y 166.991,Z 523.884,A -85,B 0,C 180,E1 -23519.637,E2 -23519.637} C_VEL
LIN {X 0,Y 171.165,Z 516.075,A -85,B 0,C 180,E1 -23522.959,E2 -23522.959} C_VEL
LIN {X 0,Y 175.99,Z 506.554,A -85,B 0,C 180,E1 -23526.087,E2 -23526.087} C_VEL
LIN {X 0,Y 180.281,Z 496.969,A -85,B 0,C 180,E1 -23528.589,E2 -23528.589} C_VEL
LIN {X 0,Y 184.861,Z 485.289,A -85,B 0,C 180,E1 -23530.98,E2 -23530.98} C_VEL
LIN {X 0,Y 188.793,Z 473.762,A -85,B 0,C 180,E1 -23532.794,E2 -23532.794} C_VEL
LIN {X 0,Y 192.429,Z 461.081,A -85,B 0,C 180,E1 -23534.305,E2 -23534.305} C_VEL
LIN {X 0,Y 195.392,Z 447.977,A -85,B 0,C 180,E1 -23535.448,E2 -23535.448} C_VEL
LIN {X 0,Y 197.669,Z 433.725,A -85,B 0,C 180,E1 -23536.291,E2 -23536.291} C_VEL
LIN {X 0,Y 199.303,Z 415.827,A -85,B 0,C 180,E1 -23536.921,E2 -23536.921} C_VEL
LIN {X 0,Y 202.687,Z 366.534,A -85,B 0,C 180,E1 -23538.489,E2 -23538.489} C_VEL
LIN {X 0,Y 197.073,Z 354.065,A -85,B 0,C 180,E1 -23541.055,E2 -23541.055} C_VEL
LIN {X 0,Y 191.734,Z 343.87,A -85,B 0,C 180,E1 -23543.68,E2 -23543.68} C_VEL
LIN {X 0,Y 186.228,Z 334.646,A -85,B 0,C 180,E1 -23546.653,E2 -23546.653} C_VEL
LIN {X 0,Y 182.755,Z 329.204,A -85,B 0,C 180,E1 -23548.725,E2 -23548.725} C_VEL
LIN {X 0,Y 180.38,Z 325.652,A -85,B 0,C 180,E1 -23550.25,E2 -23550.25} C_VEL
LIN {X 0,Y 177.112,Z 320.944,A -85,B 0,C 180,E1 -23552.53,E2 -23552.53} C_VEL
LIN {X 0,Y 173.207,Z 315.742,A -85,B 0,C 180,E1 -23555.59,E2 -23555.59} C_VEL
LIN {X 0,Y 168.613,Z 310.135,A -85,B 0,C 180,E1 -23559.888,E2 -23559.888} C_VEL
LIN {X 0,Y 164.15,Z 304.568,A -85,B 0,C 180,E1 -23565.749,E2 -23565.749} C_VEL
LIN {X 0,Y 163.692,Z 302.716,A -85,B 0,C 180,E1 -23570.112,E2 -23570.112} C_VEL
LIN {X 0,Y 163.461,Z 302.084,A -85,B 0,C 180,E1 -23572.59,E2 -23572.59} C_VEL
LIN {X 0,Y 163.445,Z 301.24,A -85,B 0,C 180,E1 -23580.001,E2 -23580.001} C_VEL
LIN {X 0,Y 163.646,Z 302.509,A -85,B 0,C 180,E1 -23587.403,E2 -23587.403} C_VEL
LIN {X 0,Y 163.889,Z 303.271,A -85,B 0,C 180,E1 -23589.878,E2 -23589.878} C_VEL
LIN {X 0,Y 164.707,Z 306.328,A -85,B 0,C 180,E1 -23596.103,E2 -23596.103} C_VEL
LIN {X 0,Y 170.478,Z 313.877,A -85,B 0,C 180,E1 -23602.897,E2 -23602.897} C_VEL
LIN {X 0,Y 175.413,Z 320.633,A -85,B 0,C 180,E1 -23607.114,E2 -23607.114} C_VEL
LIN {X 0,Y 179.275,Z 326.338,A -85,B 0,C 180,E1 -23609.921,E2 -23609.921} C_VEL
LIN {X 0,Y 182.866,Z 331.999,A -85,B 0,C 180,E1 -23612.26,E2 -23612.26} C_VEL
LIN {X 0,Y 187.864,Z 340.469,A -85,B 0,C 180,E1 -23615.186,E2 -23615.186} C_VEL
LIN {X 0,Y 192.818,Z 349.742,A -85,B 0,C 180,E1 -23617.799,E2 -23617.799} C_VEL
LIN {X 0,Y 197.641,Z 359.857,A -85,B 0,C 180,E1 -23620.13,E2 -23620.13} C_VEL
LIN {X 0,Y 201.421,Z 368.833,A -85,B 0,C 180,E1 -23621.861,E2 -23621.861} C_VEL
LIN {X 0,Y 201.915,Z 375.314,A -85,B 0,C 180,E1 -23622.347,E2 -23622.347} C_VEL
LIN {X 0,Y 198.273,Z 428.322,A -85,B 0,C 180,E1 -23623.965,E2 -23623.965} C_VEL
LIN {X 0,Y 196.432,Z 441.653,A -85,B 0,C 180,E1 -23624.677,E2 -23624.677} C_VEL
LIN {X 0,Y 193.769,Z 454.701,A -85,B 0,C 180,E1 -23625.718,E2 -23625.718} C_VEL
LIN {X 0,Y 190.762,Z 466.38,A -85,B 0,C 180,E1 -23627.034,E2 -23627.034} C_VEL
LIN {X 0,Y 186.882,Z 478.531,A -85,B 0,C 180,E1 -23628.843,E2 -23628.843} C_VEL
LIN {X 0,Y 182.688,Z 489.377,A -85,B 0,C 180,E1 -23630.955,E2 -23630.955} C_VEL
LIN {X 0,Y 177.74,Z 500.098,A -85,B 0,C 180,E1 -23633.622,E2 -23633.622} C_VEL
LIN {X 0,Y 172.944,Z 509.567,A -85,B 0,C 180,E1 -23636.729,E2 -23636.729} C_VEL
LIN {X 0,Y 168.558,Z 517.223,A -85,B 0,C 180,E1 -23639.978,E2 -23639.978} C_VEL
LIN {X 0,Y 164.52,Z 524.007,A -85,B 0,C 180,E1 -23643.779,E2 -23643.779} C_VEL
LIN {X 0,Y 160.921,Z 529.878,A -85,B 0,C 180,E1 -23648.209,E2 -23648.209} C_VEL
LIN {X 0,Y 158.457,Z 533.51,A -85,B 0,C 180,E1 -23651.913,E2 -23651.913} C_VEL
LIN {X 0,Y 156.361,Z 536.918,A -85,B 0,C 180,E1 -23657.013,E2 -23657.013} C_VEL
LIN {X 0,Y 155.66,Z 538.048,A -85,B 0,C 180,E1 -23659.595,E2 -23659.595} C_VEL
LIN {X 0,Y 154.865,Z 539.161,A -85,B 0,C 180,E1 -23664.792,E2 -23664.792} C_VEL
LIN {X 0,Y 154.835,Z 538.856,A -85,B 0,C 180,E1 -23670,E2 -23670} C_VEL
LIN {X 0,Y 155.385,Z 537.138,A -85,B 0,C 180,E1 -23675.19,E2 -23675.19} C_VEL
LIN {X 0,Y 156.737,Z 533.878,A -85,B 0,C 180,E1 -23680.332,E2 -23680.332} C_VEL
LIN {X 0,Y 158.995,Z 529.007,A -85,B 0,C 180,E1 -23685.379,E2 -23685.379} C_VEL
LIN {X 0,Y 161.442,Z 524.144,A -85,B 0,C 180,E1 -23689.056,E2 -23689.056} C_VEL
LIN {X 0,Y 165.057,Z 517.011,A -85,B 0,C 180,E1 -23693.194,E2 -23693.194} C_VEL
LIN {X 0,Y 168.728,Z 509.344,A -85,B 0,C 180,E1 -23696.6,E2 -23696.6} C_VEL
LIN {X 0,Y 172.926,Z 499.879,A -85,B 0,C 180,E1 -23699.858,E2 -23699.858} C_VEL
LIN {X 0,Y 176.862,Z 490.23,A -85,B 0,C 180,E1 -23702.442,E2 -23702.442} C_VEL
LIN {X 0,Y 180.551,Z 479.63,A -85,B 0,C 180,E1 -23704.699,E2 -23704.699} C_VEL
LIN {X 0,Y 184.168,Z 468.136,A -85,B 0,C 180,E1 -23706.555,E2 -23706.555} C_VEL
LIN {X 0,Y 187.269,Z 455.432,A -85,B 0,C 180,E1 -23708.122,E2 -23708.122} C_VEL
LIN {X 0,Y 189.791,Z 441.645,A -85,B 0,C 180,E1 -23709.34,E2 -23709.34} C_VEL
LIN {X 0,Y 191.591,Z 427.748,A -85,B 0,C 180,E1 -23710.12,E2 -23710.12} C_VEL
LIN {X 0,Y 195.156,Z 370.647,A -85,B 0,C 180,E1 -23711.959,E2 -23711.959} C_VEL
LIN {X 0,Y 194.011,Z 360.114,A -85,B 0,C 180,E1 -23712.813,E2 -23712.813} C_VEL
LIN {X 0,Y 188.851,Z 347.984,A -85,B 0,C 180,E1 -23715.056,E2 -23715.056} C_VEL
LIN {X 0,Y 183.758,Z 337.672,A -85,B 0,C 180,E1 -23717.404,E2 -23717.404} C_VEL
LIN {X 0,Y 177.996,Z 327.655,A -85,B 0,C 180,E1 -23720.279,E2 -23720.279} C_VEL
LIN {X 0,Y 174.73,Z 322.424,A -85,B 0,C 180,E1 -23722.057,E2 -23722.057} C_VEL
LIN {X 0,Y 171.88,Z 317.921,A -85,B 0,C 180,E1 -23723.727,E2 -23723.727} C_VEL
LIN {X 0,Y 167.926,Z 312.19,A -85,B 0,C 180,E1 -23726.237,E2 -23726.237} C_VEL
LIN {X 0,Y 164.351,Z 306.969,A -85,B 0,C 180,E1 -23728.949,E2 -23728.949} C_VEL
LIN {X 0,Y 163.033,Z 303.168,A -85,B 0,C 180,E1 -23733.086,E2 -23733.086} C_VEL
LIN {X 0,Y 161.961,Z 300.3,A -85,B 0,C 180,E1 -23737.011,E2 -23737.011} C_VEL
LIN {X 0,Y 160.851,Z 297.184,A -85,B 0,C 180,E1 -23742.19,E2 -23742.19} C_VEL
LIN {X 0,Y 160.461,Z 295.891,A -85,B 0,C 180,E1 -23744.763,E2 -23744.763} C_VEL
LIN {X 0,Y 159.794,Z 294.032,A -85,B 0,C 180,E1 -23749.867,E2 -23749.867} C_VEL
LIN {X 0,Y 159.473,Z 292.947,A -85,B 0,C 180,E1 -23754.942,E2 -23754.942} C_VEL
LIN {X 0,Y 159.84,Z 292.331,A -85,B 0,C 180,E1 -23759.999,E2 -23759.999} C_VEL
LIN {X 0,Y 159.794,Z 293.842,A -85,B 0,C 180,E1 -23767.581,E2 -23767.581} C_VEL
LIN {X 0,Y 160.465,Z 295.561,A -85,B 0,C 180,E1 -23772.649,E2 -23772.649} C_VEL
LIN {X 0,Y 161.274,Z 298.264,A -85,B 0,C 180,E1 -23777.76,E2 -23777.76} C_VEL
LIN {X 0,Y 162.603,Z 301.708,A -85,B 0,C 180,E1 -23782.891,E2 -23782.891} C_VEL
LIN {X 0,Y 163.564,Z 304.102,A -85,B 0,C 180,E1 -23785.617,E2 -23785.617} C_VEL
LIN {X 0,Y 167.655,Z 309.554,A -85,B 0,C 180,E1 -23788.712,E2 -23788.712} C_VEL
LIN {X 0,Y 172.524,Z 316.349,A -85,B 0,C 180,E1 -23791.804,E2 -23791.804} C_VEL
LIN {X 0,Y 176.029,Z 321.568,A -85,B 0,C 180,E1 -23793.81,E2 -23793.81} C_VEL
LIN {X 0,Y 181.53,Z 330.345,A -85,B 0,C 180,E1 -23796.673,E2 -23796.673} C_VEL
LIN {X 0,Y 187.629,Z 341.404,A -85,B 0,C 180,E1 -23799.55,E2 -23799.55} C_VEL
LIN {X 0,Y 193.319,Z 353.269,A -85,B 0,C 180,E1 -23802.044,E2 -23802.044} C_VEL
LIN {X 0,Y 196.064,Z 359.975,A -85,B 0,C 180,E1 -23803.211,E2 -23803.211} C_VEL
LIN {X 0,Y 191.383,Z 430.31,A -85,B 0,C 180,E1 -23805.593,E2 -23805.593} C_VEL
LIN {X 0,Y 189.522,Z 444.388,A -85,B 0,C 180,E1 -23806.41,E2 -23806.41} C_VEL
LIN {X 0,Y 186.848,Z 458.024,A -85,B 0,C 180,E1 -23807.571,E2 -23807.571} C_VEL
LIN {X 0,Y 183.725,Z 470.672,A -85,B 0,C 180,E1 -23809.075,E2 -23809.075} C_VEL
LIN {X 0,Y 180.061,Z 482.905,A -85,B 0,C 180,E1 -23810.997,E2 -23810.997} C_VEL
LIN {X 0,Y 176.258,Z 493.985,A -85,B 0,C 180,E1 -23813.267,E2 -23813.267} C_VEL
LIN {X 0,Y 175.885,Z 494.903,A -85,B 0,C 180,E1 -23813.48,E2 -23813.48} C_VEL
LIN {X 0,Y 173.498,Z 499.454,A -85,B 0,C 180,E1 -23814.462,E2 -23814.462} C_VEL
LIN {X 0,Y 168.112,Z 506.495,A -85,B 0,C 180,E1 -23815.94,E2 -23815.94} C_VEL
LIN {X 0,Y 162.704,Z 513.082,A -85,B 0,C 180,E1 -23817.678,E2 -23817.678} C_VEL
LIN {X 0,Y 160.34,Z 516.816,A -85,B 0,C 180,E1 -23819.061,E2 -23819.061} C_VEL
LIN {X 0,Y 156.128,Z 525.545,A -85,B 0,C 180,E1 -23823.248,E2 -23823.248} C_VEL
LIN {X 0,Y 153.296,Z 531.689,A -85,B 0,C 180,E1 -23827.065,E2 -23827.065} C_VEL
LIN {X 0,Y 150.991,Z 536.693,A -85,B 0,C 180,E1 -23830.985,E2 -23830.985} C_VEL
LIN {X 0,Y 149.196,Z 540.684,A -85,B 0,C 180,E1 -23834.985,E2 -23834.985} C_VEL
LIN {X 0,Y 148.2,Z 543.712,A -85,B 0,C 180,E1 -23839.066,E2 -23839.066} C_VEL
LIN {X 0,Y 147.605,Z 546.421,A -85,B 0,C 180,E1 -23844.536,E2 -23844.536} C_VEL
LIN {X 0,Y 147.715,Z 547.615,A -85,B 0,C 180,E1 -23850,E2 -23850} C_VEL
LIN {X 0,Y 147.607,Z 547.658,A -85,B 0,C 180,E1 -23852.729,E2 -23852.729} C_VEL
LIN {X 0,Y 147.624,Z 547.342,A -85,B 0,C 180,E1 -23855.464,E2 -23855.464} C_VEL
LIN {X 0,Y 148.224,Z 545.632,A -85,B 0,C 180,E1 -23860.933,E2 -23860.933} C_VEL
LIN {X 0,Y 149.79,Z 542.455,A -85,B 0,C 180,E1 -23866.35,E2 -23866.35} C_VEL
LIN {X 0,Y 151.852,Z 539,A -85,B 0,C 180,E1 -23870.311,E2 -23870.311} C_VEL
LIN {X 0,Y 154.89,Z 533.752,A -85,B 0,C 180,E1 -23874.842,E2 -23874.842} C_VEL
LIN {X 0,Y 158.838,Z 527.117,A -85,B 0,C 180,E1 -23879.124,E2 -23879.124} C_VEL
LIN {X 0,Y 163.693,Z 518.684,A -85,B 0,C 180,E1 -23883.189,E2 -23883.189} C_VEL
LIN {X 0,Y 168.556,Z 509.792,A -85,B 0,C 180,E1 -23886.452,E2 -23886.452} C_VEL
LIN {X 0,Y 172.956,Z 500.881,A -85,B 0,C 180,E1 -23889.037,E2 -23889.037} C_VEL
LIN {X 0,Y 177.465,Z 490.375,A -85,B 0,C 180,E1 -23891.478,E2 -23891.478} C_VEL
LIN {X 0,Y 182.092,Z 478.285,A -85,B 0,C 180,E1 -23893.621,E2 -23893.621} C_VEL
LIN {X 0,Y 185.805,Z 466.81,A -85,B 0,C 180,E1 -23895.17,E2 -23895.17} C_VEL
LIN {X 0,Y 189.087,Z 454.313,A -85,B 0,C 180,E1 -23896.449,E2 -23896.449} C_VEL
LIN {X 0,Y 191.792,Z 440.812,A -85,B 0,C 180,E1 -23897.422,E2 -23897.422} C_VEL
LIN {X 0,Y 193.566,Z 426.837,A -85,B 0,C 180,E1 -23898.1,E2 -23898.1} C_VEL
LIN {X 0,Y 197.824,Z 369.05,A -85,B 0,C 180,E1 -23899.945,E2 -23899.945} C_VEL
LIN {X 0,Y 192.737,Z 357.632,A -85,B 0,C 180,E1 -23902.438,E2 -23902.438} C_VEL
LIN {X 0,Y 187.908,Z 348.252,A -85,B 0,C 180,E1 -23904.98,E2 -23904.98} C_VEL
LIN {X 0,Y 182.814,Z 339.503,A -85,B 0,C 180,E1 -23907.928,E2 -23907.928} C_VEL
LIN {X 0,Y 178.307,Z 332.225,A -85,B 0,C 180,E1 -23910.871,E2 -23910.871} C_VEL
LIN {X 0,Y 174.802,Z 327.068,A -85,B 0,C 180,E1 -23913.431,E2 -23913.431} C_VEL
LIN {X 0,Y 171.364,Z 322.297,A -85,B 0,C 180,E1 -23916.271,E2 -23916.271} C_VEL
LIN {X 0,Y 167.018,Z 316.787,A -85,B 0,C 180,E1 -23920.536,E2 -23920.536} C_VEL
LIN {X 0,Y 162.313,Z 310.995,A -85,B 0,C 180,E1 -23926.861,E2 -23926.861} C_VEL
LIN {X 0,Y 159.597,Z 308.035,A -85,B 0,C 180,E1 -23932.727,E2 -23932.727} C_VEL
LIN {X 0,Y 158.429,Z 306.27,A -85,B 0,C 180,E1 -23940.001,E2 -23940.001} C_VEL
LIN {X 0,Y 159.057,Z 307.848,A -85,B 0,C 180,E1 -23946.343,E2 -23946.343} C_VEL
LIN {X 0,Y 160.294,Z 309.559,A -85,B 0,C 180,E1 -23950.102,E2 -23950.102} C_VEL
LIN {X 0,Y 163.591,Z 313.598,A -85,B 0,C 180,E1 -23956.056,E2 -23956.056} C_VEL
LIN {X 0,Y 168.741,Z 320.45,A -85,B 0,C 180,E1 -23962.177,E2 -23962.177} C_VEL
LIN {X 0,Y 173.181,Z 326.735,A -85,B 0,C 180,E1 -23966.182,E2 -23966.182} C_VEL
LIN {X 0,Y 176.973,Z 332.6,A -85,B 0,C 180,E1 -23969.098,E2 -23969.098} C_VEL
LIN {X 0,Y 180.156,Z 337.811,A -85,B 0,C 180,E1 -23971.289,E2 -23971.289} C_VEL
LIN {X 0,Y 184.942,Z 346.249,A -85,B 0,C 180,E1 -23974.257,E2 -23974.257} C_VEL
LIN {X 0,Y 189.311,Z 354.674,A -85,B 0,C 180,E1 -23976.693,E2 -23976.693} C_VEL
LIN {X 0,Y 193.907,Z 364.676,A -85,B 0,C 180,E1 -23979.059,E2 -23979.059} C_VEL
LIN {X 0,Y 196.836,Z 371.758,A -85,B 0,C 180,E1 -23980.491,E2 -23980.491} C_VEL
LIN {X 0,Y 197.206,Z 375.677,A -85,B 0,C 180,E1 -23980.827,E2 -23980.827} C_VEL
LIN {X 0,Y 193.469,Z 428.091,A -85,B 0,C 180,E1 -23982.439,E2 -23982.439} C_VEL
LIN {X 0,Y 191.521,Z 441.763,A -85,B 0,C 180,E1 -23983.171,E2 -23983.171} C_VEL
LIN {X 0,Y 188.756,Z 454.8,A -85,B 0,C 180,E1 -23984.215,E2 -23984.215} C_VEL
LIN {X 0,Y 185.64,Z 466.476,A -85,B 0,C 180,E1 -23985.544,E2 -23985.544} C_VEL
LIN {X 0,Y 181.884,Z 477.844,A -85,B 0,C 180,E1 -23987.238,E2 -23987.238} C_VEL
LIN {X 0,Y 177.715,Z 488.412,A -85,B 0,C 180,E1 -23989.269,E2 -23989.269} C_VEL
LIN {X 0,Y 172.985,Z 498.44,A -85,B 0,C 180,E1 -23991.716,E2 -23991.716} C_VEL
LIN {X 0,Y 168.651,Z 506.744,A -85,B 0,C 180,E1 -23994.31,E2 -23994.31} C_VEL
LIN {X 0,Y 163.938,Z 514.944,A -85,B 0,C 180,E1 -23997.597,E2 -23997.597} C_VEL
LIN {X 0,Y 159.766,Z 521.629,A -85,B 0,C 180,E1 -24001.061,E2 -24001.061} C_VEL
LIN {X 0,Y 156.294,Z 527.043,A -85,B 0,C 180,E1 -24004.712,E2 -24004.712} C_VEL
LIN {X 0,Y 153.396,Z 531.362,A -85,B 0,C 180,E1 -24008.499,E2 -24008.499} C_VEL
LIN {X 0,Y 151.701,Z 533.674,A -85,B 0,C 180,E1 -24011.077,E2 -24011.077} C_VEL
LIN {X 0,Y 149.428,Z 537.093,A -85,B 0,C 180,E1 -24016.399,E2 -24016.399} C_VEL
LIN {X 0,Y 148.672,Z 538.23,A -85,B 0,C 180,E1 -24019.101,E2 -24019.101} C_VEL
LIN {X 0,Y 147.798,Z 539.357,A -85,B 0,C 180,E1 -24024.543,E2 -24024.543} C_VEL
LIN {X 0,Y 147.748,Z 539.063,A -85,B 0,C 180,E1 -24030,E2 -24030} C_VEL
LIN {X 0,Y 148.327,Z 537.357,A -85,B 0,C 180,E1 -24035.437,E2 -24035.437} C_VEL
LIN {X 0,Y 149.774,Z 534.117,A -85,B 0,C 180,E1 -24040.818,E2 -24040.818} C_VEL
LIN {X 0,Y 152.17,Z 529.261,A -85,B 0,C 180,E1 -24046.087,E2 -24046.087} C_VEL
LIN {X 0,Y 154.766,Z 524.416,A -85,B 0,C 180,E1 -24049.912,E2 -24049.912} C_VEL
LIN {X 0,Y 158.574,Z 517.305,A -85,B 0,C 180,E1 -24054.202,E2 -24054.202} C_VEL
LIN {X 0,Y 162.4,Z 509.676,A -85,B 0,C 180,E1 -24057.724,E2 -24057.724} C_VEL
LIN {X 0,Y 166.813,Z 500.246,A -85,B 0,C 180,E1 -24061.071,E2 -24061.071} C_VEL
LIN {X 0,Y 170.944,Z 490.64,A -85,B 0,C 180,E1 -24063.712,E2 -24063.712} C_VEL
LIN {X 0,Y 174.787,Z 480.099,A -85,B 0,C 180,E1 -24066.018,E2 -24066.018} C_VEL
LIN {X 0,Y 178.665,Z 468.268,A -85,B 0,C 180,E1 -24067.97,E2 -24067.97} C_VEL
LIN {X 0,Y 181.961,Z 455.279,A -85,B 0,C 180,E1 -24069.589,E2 -24069.589} C_VEL
LIN {X 0,Y 184.516,Z 441.902,A -85,B 0,C 180,E1 -24070.782,E2 -24070.782} C_VEL
LIN {X 0,Y 186.387,Z 428.11,A -85,B 0,C 180,E1 -24071.569,E2 -24071.569} C_VEL
LIN {X 0,Y 190.045,Z 371.427,A -85,B 0,C 180,E1 -24073.439,E2 -24073.439} C_VEL
LIN {X 0,Y 189.299,Z 363.388,A -85,B 0,C 180,E1 -24074.095,E2 -24074.095} C_VEL
LIN {X 0,Y 184.738,Z 352.362,A -85,B 0,C 180,E1 -24076.219,E2 -24076.219} C_VEL
LIN {X 0,Y 180.041,Z 342.545,A -85,B 0,C 180,E1 -24078.531,E2 -24078.531} C_VEL
LIN {X 0,Y 174.663,Z 332.918,A -85,B 0,C 180,E1 -24081.388,E2 -24081.388} C_VEL
LIN {X 0,Y 171.636,Z 327.902,A -85,B 0,C 180,E1 -24083.142,E2 -24083.142} C_VEL
LIN {X 0,Y 168.842,Z 323.393,A -85,B 0,C 180,E1 -24084.884,E2 -24084.884} C_VEL
LIN {X 0,Y 165.318,Z 318.085,A -85,B 0,C 180,E1 -24087.268,E2 -24087.268} C_VEL
LIN {X 0,Y 161.446,Z 312.596,A -85,B 0,C 180,E1 -24090.204,E2 -24090.204} C_VEL
LIN {X 0,Y 157.002,Z 306.497,A -85,B 0,C 180,E1 -24094.44,E2 -24094.44} C_VEL
LIN {X 0,Y 155.891,Z 303.444,A -85,B 0,C 180,E1 -24098.858,E2 -24098.858} C_VEL
LIN {X 0,Y 154.978,Z 300.627,A -85,B 0,C 180,E1 -24104.21,E2 -24104.21} C_VEL
LIN {X 0,Y 154.337,Z 298.654,A -85,B 0,C 180,E1 -24109.504,E2 -24109.504} C_VEL
LIN {X 0,Y 154.02,Z 297.51,A -85,B 0,C 180,E1 -24114.763,E2 -24114.763} C_VEL
LIN {X 0,Y 154.372,Z 296.887,A -85,B 0,C 180,E1 -24119.999,E2 -24119.999} C_VEL
LIN {X 0,Y 154.105,Z 297.849,A -85,B 0,C 180,E1 -24125.232,E2 -24125.232} C_VEL
LIN {X 0,Y 154.618,Z 299.232,A -85,B 0,C 180,E1 -24130.475,E2 -24130.475} C_VEL
LIN {X 0,Y 154.956,Z 300.286,A -85,B 0,C 180,E1 -24133.106,E2 -24133.106} C_VEL
LIN {X 0,Y 156.339,Z 304.2,A -85,B 0,C 180,E1 -24140.044,E2 -24140.044} C_VEL
LIN {X 0,Y 160.752,Z 309.832,A -85,B 0,C 180,E1 -24144.366,E2 -24144.366} C_VEL
LIN {X 0,Y 165.985,Z 316.911,A -85,B 0,C 180,E1 -24148.36,E2 -24148.36} C_VEL
LIN {X 0,Y 169.7,Z 322.206,A -85,B 0,C 180,E1 -24150.819,E2 -24150.819} C_VEL
LIN {X 0,Y 173.16,Z 327.481,A -85,B 0,C 180,E1 -24152.909,E2 -24152.909} C_VEL
LIN {X 0,Y 178.278,Z 335.976,A -85,B 0,C 180,E1 -24155.727,E2 -24155.727} C_VEL
LIN {X 0,Y 183.675,Z 346.062,A -85,B 0,C 180,E1 -24158.434,E2 -24158.434} C_VEL
LIN {X 0,Y 189.095,Z 357.75,A -85,B 0,C 180,E1 -24160.968,E2 -24160.968} C_VEL
LIN {X 0,Y 190.938,Z 362.306,A -85,B 0,C 180,E1 -24161.804,E2 -24161.804} C_VEL
LIN {X 0,Y 186.247,Z 429.775,A -85,B 0,C 180,E1 -24164.098,E2 -24164.098} C_VEL
LIN {X 0,Y 184.286,Z 444.199,A -85,B 0,C 180,E1 -24164.936,E2 -24164.936} C_VEL
LIN {X 0,Y 181.616,Z 457.296,A -85,B 0,C 180,E1 -24166.043,E2 -24166.043} C_VEL
LIN {X 0,Y 178.393,Z 470.086,A -85,B 0,C 180,E1 -24167.573,E2 -24167.573} C_VEL
LIN {X 0,Y 174.559,Z 482.424,A -85,B 0,C 180,E1 -24169.519,E2 -24169.519} C_VEL
LIN {X 0,Y 170.604,Z 493.583,A -85,B 0,C 180,E1 -24171.836,E2 -24171.836} C_VEL
LIN {X 0,Y 166.36,Z 503.75,A -85,B 0,C 180,E1 -24174.489,E2 -24174.489} C_VEL
LIN {X 0,Y 161.738,Z 513.763,A -85,B 0,C 180,E1 -24177.84,E2 -24177.84} C_VEL
LIN {X 0,Y 160.34,Z 516.816,A -85,B 0,C 180,E1 -24179.061,E2 -24179.061} C_VEL
LIN {X 0,Y 158.03,Z 520.425,A -85,B 0,C 180,E1 -24180.543,E2 -24180.543} C_VEL
LIN {X 0,Y 152.816,Z 525.865,A -85,B 0,C 180,E1 -24182.905,E2 -24182.905} C_VEL
LIN {X 0,Y 147.754,Z 530.773,A -85,B 0,C 180,E1 -24185.558,E2 -24185.558} C_VEL
LIN {X 0,Y 145.75,Z 533.412,A -85,B 0,C 180,E1 -24187.467,E2 -24187.467} C_VEL
LIN {X 0,Y 143.522,Z 537.891,A -85,B 0,C 180,E1 -24191.441,E2 -24191.441} C_VEL
LIN {X 0,Y 141.854,Z 541.536,A -85,B 0,C 180,E1 -24195.658,E2 -24195.658} C_VEL
LIN {X 0,Y 140.743,Z 545.036,A -85,B 0,C 180,E1 -24201.385,E2 -24201.385} C_VEL
LIN {X 0,Y 140.526,Z 546.207,A -85,B 0,C 180,E1 -24204.26,E2 -24204.26} C_VEL
LIN {X 0,Y 140.627,Z 547.413,A -85,B 0,C 180,E1 -24210,E2 -24210} C_VEL
LIN {X 0,Y 140.503,Z 547.462,A -85,B 0,C 180,E1 -24212.867,E2 -24212.867} C_VEL
LIN {X 0,Y 140.758,Z 546.48,A -85,B 0,C 180,E1 -24218.615,E2 -24218.615} C_VEL
LIN {X 0,Y 141.935,Z 544.054,A -85,B 0,C 180,E1 -24224.334,E2 -24224.334} C_VEL
LIN {X 0,Y 143.659,Z 541.218,A -85,B 0,C 180,E1 -24228.541,E2 -24228.541} C_VEL
LIN {X 0,Y 146.965,Z 536.042,A -85,B 0,C 180,E1 -24233.983,E2 -24233.983} C_VEL
LIN {X 0,Y 150.111,Z 530.953,A -85,B 0,C 180,E1 -24237.916,E2 -24237.916} C_VEL
LIN {X 0,Y 154.744,Z 523.605,A -85,B 0,C 180,E1 -24242.252,E2 -24242.252} C_VEL
LIN {X 0,Y 159.394,Z 515.813,A -85,B 0,C 180,E1 -24245.747,E2 -24245.747} C_VEL
LIN {X 0,Y 164.695,Z 506.308,A -85,B 0,C 180,E1 -24249.007,E2 -24249.007} C_VEL
LIN {X 0,Y 169.727,Z 495.862,A -85,B 0,C 180,E1 -24251.813,E2 -24251.813} C_VEL
LIN {X 0,Y 174.376,Z 485.059,A -85,B 0,C 180,E1 -24254.045,E2 -24254.045} C_VEL
LIN {X 0,Y 178.647,Z 473.533,A -85,B 0,C 180,E1 -24255.885,E2 -24255.885} C_VEL
LIN {X 0,Y 182.534,Z 460.842,A -85,B 0,C 180,E1 -24257.421,E2 -24257.421} C_VEL
LIN {X 0,Y 185.701,Z 447.698,A -85,B 0,C 180,E1 -24258.574,E2 -24258.574} C_VEL
LIN {X 0,Y 188.049,Z 434.146,A -85,B 0,C 180,E1 -24259.377,E2 -24259.377} C_VEL
LIN {X 0,Y 189.643,Z 418.662,A -85,B 0,C 180,E1 -24259.94,E2 -24259.94} C_VEL
LIN {X 0,Y 193.078,Z 371.532,A -85,B 0,C 180,E1 -24261.481,E2 -24261.481} C_VEL
LIN {X 0,Y 188.247,Z 360.571,A -85,B 0,C 180,E1 -24264.041,E2 -24264.041} C_VEL
LIN {X 0,Y 183.077,Z 350.553,A -85,B 0,C 180,E1 -24267.001,E2 -24267.001} C_VEL
LIN {X 0,Y 177.81,Z 341.46,A -85,B 0,C 180,E1 -24270.394,E2 -24270.394} C_VEL
LIN {X 0,Y 174.603,Z 336.452,A -85,B 0,C 180,E1 -24272.711,E2 -24272.711} C_VEL
LIN {X 0,Y 172.515,Z 333.201,A -85,B 0,C 180,E1 -24274.37,E2 -24274.37} C_VEL
LIN {X 0,Y 169.31,Z 328.579,A -85,B 0,C 180,E1 -24277.18,E2 -24277.18} C_VEL
LIN {X 0,Y 165.292,Z 323.272,A -85,B 0,C 180,E1 -24281.371,E2 -24281.371} C_VEL
LIN {X 0,Y 161.067,Z 317.826,A -85,B 0,C 180,E1 -24287.399,E2 -24287.399} C_VEL
LIN {X 0,Y 158.61,Z 315,A -85,B 0,C 180,E1 -24293.002,E2 -24293.002} C_VEL
LIN {X 0,Y 157.519,Z 313.322,A -85,B 0,C 180,E1 -24300.001,E2 -24300.001} C_VEL
LIN {X 0,Y 158.368,Z 315.125,A -85,B 0,C 180,E1 -24307.011,E2 -24307.011} C_VEL
LIN {X 0,Y 159.824,Z 317.38,A -85,B 0,C 180,E1 -24311.093,E2 -24311.093} C_VEL
LIN {X 0,Y 162.316,Z 320.467,A -85,B 0,C 180,E1 -24315.541,E2 -24315.541} C_VEL
LIN {X 0,Y 166.967,Z 326.908,A -85,B 0,C 180,E1 -24321.369,E2 -24321.369} C_VEL
LIN {X 0,Y 171.117,Z 333.06,A -85,B 0,C 180,E1 -24325.334,E2 -24325.334} C_VEL
LIN {X 0,Y 174.724,Z 338.92,A -85,B 0,C 180,E1 -24328.269,E2 -24328.269} C_VEL
LIN {X 0,Y 177.44,Z 343.56,A -85,B 0,C 180,E1 -24330.25,E2 -24330.25} C_VEL
LIN {X 0,Y 181.666,Z 351.198,A -85,B 0,C 180,E1 -24333.042,E2 -24333.042} C_VEL
LIN {X 0,Y 186.611,Z 361.197,A -85,B 0,C 180,E1 -24335.962,E2 -24335.962} C_VEL
LIN {X 0,Y 191.385,Z 372.228,A -85,B 0,C 180,E1 -24338.547,E2 -24338.547} C_VEL
LIN {X 0,Y 192.467,Z 374.988,A -85,B 0,C 180,E1 -24339.11,E2 -24339.11} C_VEL
LIN {X 0,Y 192.457,Z 378.663,A -85,B 0,C 180,E1 -24339.314,E2 -24339.314} C_VEL
LIN {X 0,Y 188.786,Z 428.063,A -85,B 0,C 180,E1 -24340.845,E2 -24340.845} C_VEL
LIN {X 0,Y 186.747,Z 441.875,A -85,B 0,C 180,E1 -24341.586,E2 -24341.586} C_VEL
LIN {X 0,Y 183.882,Z 454.9,A -85,B 0,C 180,E1 -24342.631,E2 -24342.631} C_VEL
LIN {X 0,Y 180.648,Z 466.573,A -85,B 0,C 180,E1 -24343.969,E2 -24343.969} C_VEL
LIN {X 0,Y 176.452,Z 478.702,A -85,B 0,C 180,E1 -24345.803,E2 -24345.803} C_VEL
LIN {X 0,Y 171.898,Z 489.587,A -85,B 0,C 180,E1 -24347.973,E2 -24347.973} C_VEL
LIN {X 0,Y 166.513,Z 500.322,A -85,B 0,C 180,E1 -24350.721,E2 -24350.721} C_VEL
LIN {X 0,Y 161.222,Z 509.81,A -85,B 0,C 180,E1 -24353.95,E2 -24353.95} C_VEL
LIN {X 0,Y 156.404,Z 517.489,A -85,B 0,C 180,E1 -24357.37,E2 -24357.37} C_VEL
LIN {X 0,Y 152.159,Z 523.912,A -85,B 0,C 180,E1 -24361.14,E2 -24361.14} C_VEL
LIN {X 0,Y 148.758,Z 528.776,A -85,B 0,C 180,E1 -24364.837,E2 -24364.837} C_VEL
LIN {X 0,Y 145.876,Z 532.742,A -85,B 0,C 180,E1 -24368.818,E2 -24368.818} C_VEL
LIN {X 0,Y 143.593,Z 535.747,A -85,B 0,C 180,E1 -24372.923,E2 -24372.923} C_VEL
LIN {X 0,Y 141.682,Z 538.413,A -85,B 0,C 180,E1 -24378.556,E2 -24378.556} C_VEL
LIN {X 0,Y 140.725,Z 539.553,A -85,B 0,C 180,E1 -24384.268,E2 -24384.268} C_VEL
LIN {X 0,Y 140.652,Z 539.27,A -85,B 0,C 180,E1 -24390,E2 -24390} C_VEL
LIN {X 0,Y 141.264,Z 537.576,A -85,B 0,C 180,E1 -24395.71,E2 -24395.71} C_VEL
LIN {X 0,Y 141.893,Z 536.172,A -85,B 0,C 180,E1 -24398.545,E2 -24398.545} C_VEL
LIN {X 0,Y 143.956,Z 532.144,A -85,B 0,C 180,E1 -24404.128,E2 -24404.128} C_VEL
LIN {X 0,Y 146.237,Z 528.029,A -85,B 0,C 180,E1 -24408.202,E2 -24408.202} C_VEL
LIN {X 0,Y 149.179,Z 522.842,A -85,B 0,C 180,E1 -24412.141,E2 -24412.141} C_VEL
LIN {X 0,Y 153.419,Z 515.209,A -85,B 0,C 180,E1 -24416.528,E2 -24416.528} C_VEL
LIN {X 0,Y 157.696,Z 507.072,A -85,B 0,C 180,E1 -24420.09,E2 -24420.09} C_VEL
LIN {X 0,Y 161.61,Z 498.849,A -85,B 0,C 180,E1 -24422.928,E2 -24422.928} C_VEL
LIN {X 0,Y 165.992,Z 488.93,A -85,B 0,C 180,E1 -24425.602,E2 -24425.602} C_VEL
LIN {X 0,Y 169.637,Z 479.281,A -85,B 0,C 180,E1 -24427.667,E2 -24427.667} C_VEL
LIN {X 0,Y 173.138,Z 468.817,A -85,B 0,C 180,E1 -24429.412,E2 -24429.412} C_VEL
LIN {X 0,Y 176.591,Z 456.022,A -85,B 0,C 180,E1 -24431.045,E2 -24431.045} C_VEL
LIN {X 0,Y 179.223,Z 442.893,A -85,B 0,C 180,E1 -24432.258,E2 -24432.258} C_VEL
LIN {X 0,Y 181.146,Z 429.605,A -85,B 0,C 180,E1 -24433.054,E2 -24433.054} C_VEL
LIN {X 0,Y 183.213,Z 402.177,A -85,B 0,C 180,E1 -24433.988,E2 -24433.988} C_VEL
LIN {X 0,Y 185.122,Z 372.424,A -85,B 0,C 180,E1 -24434.972,E2 -24434.972} C_VEL
LIN {X 0,Y 184.567,Z 366.27,A -85,B 0,C 180,E1 -24435.5,E2 -24435.5} C_VEL
LIN {X 0,Y 180.003,Z 355.085,A -85,B 0,C 180,E1 -24437.798,E2 -24437.798} C_VEL
LIN {X 0,Y 175.41,Z 345.602,A -85,B 0,C 180,E1 -24440.237,E2 -24440.237} C_VEL
LIN {X 0,Y 171.247,Z 337.93,A -85,B 0,C 180,E1 -24442.63,E2 -24442.63} C_VEL
LIN {X 0,Y 166.49,Z 329.737,A -85,B 0,C 180,E1 -24445.672,E2 -24445.672} C_VEL
LIN {X 0,Y 162.732,Z 323.954,A -85,B 0,C 180,E1 -24448.354,E2 -24448.354} C_VEL
LIN {X 0,Y 158.997,Z 318.543,A -85,B 0,C 180,E1 -24451.375,E2 -24451.375} C_VEL
LIN {X 0,Y 154.554,Z 312.527,A -85,B 0,C 180,E1 -24455.645,E2 -24455.645} C_VEL
LIN {X 0,Y 149.81,Z 306.237,A -85,B 0,C 180,E1 -24461.998,E2 -24461.998} C_VEL
LIN {X 0,Y 149.103,Z 304.204,A -85,B 0,C 180,E1 -24466.368,E2 -24466.368} C_VEL
LIN {X 0,Y 148.668,Z 302.581,A -85,B 0,C 180,E1 -24471.846,E2 -24471.846} C_VEL
LIN {X 0,Y 148.683,Z 301.663,A -85,B 0,C 180,E1 -24477.29,E2 -24477.29} C_VEL
LIN {X 0,Y 148.905,Z 301.443,A -85,B 0,C 180,E1 -24479.999,E2 -24479.999} C_VEL
LIN {X 0,Y 148.776,Z 302.833,A -85,B 0,C 180,E1 -24487.255,E2 -24487.255} C_VEL
LIN {X 0,Y 149.548,Z 304.783,A -85,B 0,C 180,E1 -24492.725,E2 -24492.725} C_VEL
LIN {X 0,Y 154.92,Z 311.501,A -85,B 0,C 180,E1 -24499.891,E2 -24499.891} C_VEL
LIN {X 0,Y 159.495,Z 317.299,A -85,B 0,C 180,E1 -24504.204,E2 -24504.204} C_VEL
LIN {X 0,Y 163.64,Z 323.18,A -85,B 0,C 180,E1 -24507.495,E2 -24507.495} C_VEL
LIN {X 0,Y 167.259,Z 328.529,A -85,B 0,C 180,E1 -24510.018,E2 -24510.018} C_VEL
LIN {X 0,Y 170.46,Z 333.678,A -85,B 0,C 180,E1 -24512.061,E2 -24512.061} C_VEL
LIN {X 0,Y 175.632,Z 342.561,A -85,B 0,C 180,E1 -24515.049,E2 -24515.049} C_VEL
LIN {X 0,Y 180.867,Z 352.962,A -85,B 0,C 180,E1 -24517.82,E2 -24517.82} C_VEL
LIN {X 0,Y 185.859,Z 364.547,A -85,B 0,C 180,E1 -24520.29,E2 -24520.29} C_VEL
LIN {X 0,Y 182.226,Z 417.166,A -85,B 0,C 180,E1 -24522.094,E2 -24522.094} C_VEL
LIN {X 0,Y 180.662,Z 434.077,A -85,B 0,C 180,E1 -24522.756,E2 -24522.756} C_VEL
LIN {X 0,Y 178.499,Z 447.808,A -85,B 0,C 180,E1 -24523.659,E2 -24523.659} C_VEL
LIN {X 0,Y 175.822,Z 459.964,A -85,B 0,C 180,E1 -24524.806,E2 -24524.806} C_VEL
LIN {X 0,Y 172.171,Z 472.896,A -85,B 0,C 180,E1 -24526.463,E2 -24526.463} C_VEL
LIN {X 0,Y 168.27,Z 484.484,A -85,B 0,C 180,E1 -24528.434,E2 -24528.434} C_VEL
LIN {X 0,Y 163.648,Z 496.416,A -85,B 0,C 180,E1 -24531.092,E2 -24531.092} C_VEL
LIN {X 0,Y 158.913,Z 506.99,A -85,B 0,C 180,E1 -24534.128,E2 -24534.128} C_VEL
LIN {X 0,Y 154.308,Z 516.391,A -85,B 0,C 180,E1 -24537.646,E2 -24537.646} C_VEL
LIN {X 0,Y 150.353,Z 524.119,A -85,B 0,C 180,E1 -24541.373,E2 -24541.373} C_VEL
LIN {X 0,Y 147.37,Z 530.034,A -85,B 0,C 180,E1 -24544.97,E2 -24544.97} C_VEL
LIN {X 0,Y 145.75,Z 533.412,A -85,B 0,C 180,E1 -24547.467,E2 -24547.467} C_VEL
LIN {X 0,Y 143.853,Z 535.891,A -85,B 0,C 180,E1 -24549.466,E2 -24549.466} C_VEL
LIN {X 0,Y 137.534,Z 540.603,A -85,B 0,C 180,E1 -24554.118,E2 -24554.118} C_VEL
LIN {X 0,Y 134.693,Z 542.749,A -85,B 0,C 180,E1 -24557.095,E2 -24557.095} C_VEL
LIN {X 0,Y 134.026,Z 543.662,A -85,B 0,C 180,E1 -24558.706,E2 -24558.706} C_VEL
LIN {X 0,Y 133.442,Z 545.992,A -85,B 0,C 180,E1 -24563.954,E2 -24563.954} C_VEL
LIN {X 0,Y 133.394,Z 546.785,A -85,B 0,C 180,E1 -24566.98,E2 -24566.98} C_VEL
LIN {X 0,Y 133.53,Z 547.212,A -85,B 0,C 180,E1 -24570,E2 -24570} C_VEL
LIN {X 0,Y 133.405,Z 547.265,A -85,B 0,C 180,E1 -24573.02,E2 -24573.02} C_VEL
LIN {X 0,Y 133.71,Z 546.293,A -85,B 0,C 180,E1 -24579.073,E2 -24579.073} C_VEL
LIN {X 0,Y 135.01,Z 543.877,A -85,B 0,C 180,E1 -24585.086,E2 -24585.086} C_VEL
LIN {X 0,Y 137.694,Z 539.941,A -85,B 0,C 180,E1 -24590.933,E2 -24590.933} C_VEL
LIN {X 0,Y 140.431,Z 535.884,A -85,B 0,C 180,E1 -24595.175,E2 -24595.175} C_VEL
LIN {X 0,Y 143.816,Z 530.804,A -85,B 0,C 180,E1 -24599.253,E2 -24599.253} C_VEL
LIN {X 0,Y 148.748,Z 523.466,A -85,B 0,C 180,E1 -24603.721,E2 -24603.721} C_VEL
LIN {X 0,Y 153.646,Z 515.682,A -85,B 0,C 180,E1 -24607.306,E2 -24607.306} C_VEL
LIN {X 0,Y 159.228,Z 506.186,A -85,B 0,C 180,E1 -24610.619,E2 -24610.619} C_VEL
LIN {X 0,Y 164.177,Z 496.419,A -85,B 0,C 180,E1 -24613.305,E2 -24613.305} C_VEL
LIN {X 0,Y 169.333,Z 484.945,A -85,B 0,C 180,E1 -24615.72,E2 -24615.72} C_VEL
LIN {X 0,Y 173.779,Z 473.42,A -85,B 0,C 180,E1 -24617.566,E2 -24617.566} C_VEL
LIN {X 0,Y 177.817,Z 460.724,A -85,B 0,C 180,E1 -24619.102,E2 -24619.102} C_VEL
LIN {X 0,Y 181.081,Z 447.559,A -85,B 0,C 180,E1 -24620.258,E2 -24620.258} C_VEL
LIN {X 0,Y 183.49,Z 434.075,A -85,B 0,C 180,E1 -24621.055,E2 -24621.055} C_VEL
LIN {X 0,Y 185.206,Z 417.735,A -85,B 0,C 180,E1 -24621.642,E2 -24621.642} C_VEL
LIN {X 0,Y 188.502,Z 374.146,A -85,B 0,C 180,E1 -24623.075,E2 -24623.075} C_VEL
LIN {X 0,Y 184.245,Z 364.344,A -85,B 0,C 180,E1 -24625.514,E2 -24625.514} C_VEL
LIN {X 0,Y 179.423,Z 354.823,A -85,B 0,C 180,E1 -24628.497,E2 -24628.497} C_VEL
LIN {X 0,Y 174.959,Z 346.895,A -85,B 0,C 180,E1 -24631.592,E2 -24631.592} C_VEL
LIN {X 0,Y 172.347,Z 342.611,A -85,B 0,C 180,E1 -24633.604,E2 -24633.604} C_VEL
LIN {X 0,Y 170.001,Z 338.918,A -85,B 0,C 180,E1 -24635.582,E2 -24635.582} C_VEL
LIN {X 0,Y 167.306,Z 334.867,A -85,B 0,C 180,E1 -24638.112,E2 -24638.112} C_VEL
LIN {X 0,Y 163.773,Z 329.961,A -85,B 0,C 180,E1 -24642.023,E2 -24642.023} C_VEL
LIN {X 0,Y 159.849,Z 324.652,A -85,B 0,C 180,E1 -24647.946,E2 -24647.946} C_VEL
LIN {X 0,Y 157.644,Z 321.996,A -85,B 0,C 180,E1 -24653.28,E2 -24653.28} C_VEL
LIN {X 0,Y 156.652,Z 320.384,A -85,B 0,C 180,E1 -24660.001,E2 -24660.001} C_VEL
LIN {X 0,Y 157.506,Z 322.239,A -85,B 0,C 180,E1 -24667.049,E2 -24667.049} C_VEL
LIN {X 0,Y 160.674,Z 326.647,A -85,B 0,C 180,E1 -24674.366,E2 -24674.366} C_VEL
LIN {X 0,Y 165.232,Z 333.394,A -85,B 0,C 180,E1 -24680.554,E2 -24680.554} C_VEL
LIN {X 0,Y 169.105,Z 339.413,A -85,B 0,C 180,E1 -24684.479,E2 -24684.479} C_VEL
LIN {X 0,Y 172.202,Z 344.665,A -85,B 0,C 180,E1 -24687.163,E2 -24687.163} C_VEL
LIN {X 0,Y 174.878,Z 349.425,A -85,B 0,C 180,E1 -24689.245,E2 -24689.245} C_VEL
LIN {X 0,Y 178.957,Z 357.229,A -85,B 0,C 180,E1 -24692.105,E2 -24692.105} C_VEL
LIN {X 0,Y 182.823,Z 365.263,A -85,B 0,C 180,E1 -24694.543,E2 -24694.543} C_VEL
LIN {X 0,Y 186.757,Z 374.604,A -85,B 0,C 180,E1 -24696.856,E2 -24696.856} C_VEL
LIN {X 0,Y 188.066,Z 377.879,A -85,B 0,C 180,E1 -24697.587,E2 -24697.587} C_VEL
LIN {X 0,Y 184.232,Z 428.243,A -85,B 0,C 180,E1 -24699.182,E2 -24699.182} C_VEL
LIN {X 0,Y 182.117,Z 441.986,A -85,B 0,C 180,E1 -24699.917,E2 -24699.917} C_VEL
LIN {X 0,Y 179.15,Z 454.998,A -85,B 0,C 180,E1 -24700.961,E2 -24700.961} C_VEL
LIN {X 0,Y 175.782,Z 466.669,A -85,B 0,C 180,E1 -24702.299,E2 -24702.299} C_VEL
LIN {X 0,Y 171.551,Z 478.493,A -85,B 0,C 180,E1 -24704.093,E2 -24704.093} C_VEL
LIN {X 0,Y 166.694,Z 489.692,A -85,B 0,C 180,E1 -24706.34,E2 -24706.34} C_VEL
LIN {X 0,Y 161.083,Z 500.434,A -85,B 0,C 180,E1 -24709.123,E2 -24709.123} C_VEL
LIN {X 0,Y 155.518,Z 509.931,A -85,B 0,C 180,E1 -24712.406,E2 -24712.406} C_VEL
LIN {X 0,Y 150.464,Z 517.621,A -85,B 0,C 180,E1 -24715.91,E2 -24715.91} C_VEL
LIN {X 0,Y 146.071,Z 523.876,A -85,B 0,C 180,E1 -24719.656,E2 -24719.656} C_VEL
LIN {X 0,Y 142.336,Z 528.927,A -85,B 0,C 180,E1 -24723.616,E2 -24723.616} C_VEL
LIN {X 0,Y 139.27,Z 532.901,A -85,B 0,C 180,E1 -24727.761,E2 -24727.761} C_VEL
LIN {X 0,Y 136.781,Z 535.916,A -85,B 0,C 180,E1 -24732.044,E2 -24732.044} C_VEL
LIN {X 0,Y 134.718,Z 538.594,A -85,B 0,C 180,E1 -24737.956,E2 -24737.956} C_VEL
LIN {X 0,Y 133.656,Z 539.749,A -85,B 0,C 180,E1 -24743.963,E2 -24743.963} C_VEL
LIN {X 0,Y 133.575,Z 539.477,A -85,B 0,C 180,E1 -24750,E2 -24750} C_VEL
LIN {X 0,Y 134.215,Z 537.795,A -85,B 0,C 180,E1 -24756.011,E2 -24756.011} C_VEL
LIN {X 0,Y 134.881,Z 536.402,A -85,B 0,C 180,E1 -24758.993,E2 -24758.993} C_VEL
LIN {X 0,Y 136.461,Z 533.551,A -85,B 0,C 180,E1 -24763.4,E2 -24763.4} C_VEL
LIN {X 0,Y 138.602,Z 529.769,A -85,B 0,C 180,E1 -24767.712,E2 -24767.712} C_VEL
LIN {X 0,Y 141.542,Z 524.958,A -85,B 0,C 180,E1 -24771.863,E2 -24771.863} C_VEL
LIN {X 0,Y 145.753,Z 517.889,A -85,B 0,C 180,E1 -24776.488,E2 -24776.488} C_VEL
LIN {X 0,Y 149.995,Z 510.325,A -85,B 0,C 180,E1 -24780.244,E2 -24780.244} C_VEL
LIN {X 0,Y 154.86,Z 500.978,A -85,B 0,C 180,E1 -24783.775,E2 -24783.775} C_VEL
LIN {X 0,Y 159.383,Z 491.459,A -85,B 0,C 180,E1 -24786.532,E2 -24786.532} C_VEL
LIN {X 0,Y 163.571,Z 481.034,A -85,B 0,C 180,E1 -24788.93,E2 -24788.93} C_VEL
LIN {X 0,Y 167.818,Z 469.108,A -85,B 0,C 180,E1 -24790.985,E2 -24790.985} C_VEL
LIN {X 0,Y 171.341,Z 456.759,A -85,B 0,C 180,E1 -24792.592,E2 -24792.592} C_VEL
LIN {X 0,Y 174.075,Z 443.879,A -85,B 0,C 180,E1 -24793.816,E2 -24793.816} C_VEL
LIN {X 0,Y 176.186,Z 429.991,A -85,B 0,C 180,E1 -24794.673,E2 -24794.673} C_VEL
LIN {X 0,Y 178.032,Z 406.801,A -85,B 0,C 180,E1 -24795.492,E2 -24795.492} C_VEL
LIN {X 0,Y 180.327,Z 373.389,A -85,B 0,C 180,E1 -24796.594,E2 -24796.594} C_VEL
LIN {X 0,Y 179.946,Z 369.216,A -85,B 0,C 180,E1 -24796.977,E2 -24796.977} C_VEL
LIN {X 0,Y 175.197,Z 357.497,A -85,B 0,C 180,E1 -24799.563,E2 -24799.563} C_VEL
LIN {X 0,Y 170.711,Z 348.142,A -85,B 0,C 180,E1 -24802.178,E2 -24802.178} C_VEL
LIN {X 0,Y 166.199,Z 339.797,A -85,B 0,C 180,E1 -24805.058,E2 -24805.058} C_VEL
LIN {X 0,Y 162.804,Z 334.029,A -85,B 0,C 180,E1 -24807.458,E2 -24807.458} C_VEL
LIN {X 0,Y 160.237,Z 329.849,A -85,B 0,C 180,E1 -24809.453,E2 -24809.453} C_VEL
LIN {X 0,Y 156.897,Z 324.803,A -85,B 0,C 180,E1 -24812.333,E2 -24812.333} C_VEL
LIN {X 0,Y 152.768,Z 318.972,A -85,B 0,C 180,E1 -24816.554,E2 -24816.554} C_VEL
LIN {X 0,Y 147.963,Z 312.585,A -85,B 0,C 180,E1 -24823.232,E2 -24823.232} C_VEL
LIN {X 0,Y 144.858,Z 308.896,A -85,B 0,C 180,E1 -24830.575,E2 -24830.575} C_VEL
LIN {X 0,Y 143.996,Z 307.014,A -85,B 0,C 180,E1 -24837.202,E2 -24837.202} C_VEL
LIN {X 0,Y 144.174,Z 306.812,A -85,B 0,C 180,E1 -24840.348,E2 -24840.348} C_VEL
LIN {X 0,Y 147.282,Z 310.752,A -85,B 0,C 180,E1 -24850.655,E2 -24850.655} C_VEL
LIN {X 0,Y 148.49,Z 312.234,A -85,B 0,C 180,E1 -24852.817,E2 -24852.817} C_VEL
LIN {X 0,Y 153.136,Z 317.979,A -85,B 0,C 180,E1 -24859.031,E2 -24859.031} C_VEL
LIN {X 0,Y 157.443,Z 323.696,A -85,B 0,C 180,E1 -24863.338,E2 -24863.338} C_VEL
LIN {X 0,Y 161.232,Z 329.288,A -85,B 0,C 180,E1 -24866.526,E2 -24866.526} C_VEL
LIN {X 0,Y 164.566,Z 334.441,A -85,B 0,C 180,E1 -24868.998,E2 -24868.998} C_VEL
LIN {X 0,Y 167.769,Z 339.764,A -85,B 0,C 180,E1 -24871.161,E2 -24871.161} C_VEL
LIN {X 0,Y 172.511,Z 348.27,A -85,B 0,C 180,E1 -24874.067,E2 -24874.067} C_VEL
LIN {X 0,Y 177.331,Z 358.302,A -85,B 0,C 180,E1 -24876.79,E2 -24876.79} C_VEL
LIN {X 0,Y 180.992,Z 366.944,A -85,B 0,C 180,E1 -24878.729,E2 -24878.729} C_VEL
LIN {X 0,Y 176.2,Z 430.424,A -85,B 0,C 180,E1 -24880.945,E2 -24880.945} C_VEL
LIN {X 0,Y 174.24,Z 443.822,A -85,B 0,C 180,E1 -24881.739,E2 -24881.739} C_VEL
LIN {X 0,Y 171.08,Z 458.112,A -85,B 0,C 180,E1 -24882.969,E2 -24882.969} C_VEL
LIN {X 0,Y 167.617,Z 470.689,A -85,B 0,C 180,E1 -24884.539,E2 -24884.539} C_VEL
LIN {X 0,Y 163.451,Z 482.835,A -85,B 0,C 180,E1 -24886.532,E2 -24886.532} C_VEL
LIN {X 0,Y 159.141,Z 493.856,A -85,B 0,C 180,E1 -24888.936,E2 -24888.936} C_VEL
LIN {X 0,Y 154.965,Z 503.028,A -85,B 0,C 180,E1 -24891.422,E2 -24891.422} C_VEL
LIN {X 0,Y 149.812,Z 513.106,A -85,B 0,C 180,E1 -24894.924,E2 -24894.924} C_VEL
LIN {X 0,Y 145.422,Z 521.388,A -85,B 0,C 180,E1 -24898.7,E2 -24898.7} C_VEL
LIN {X 0,Y 141.17,Z 529.232,A -85,B 0,C 180,E1 -24903.382,E2 -24903.382} C_VEL
LIN {X 0,Y 138.34,Z 534.622,A -85,B 0,C 180,E1 -24907.604,E2 -24907.604} C_VEL
LIN {X 0,Y 136.06,Z 538.95,A -85,B 0,C 180,E1 -24911.946,E2 -24911.946} C_VEL
LIN {X 0,Y 134.195,Z 543.247,A -85,B 0,C 180,E1 -24917.908,E2 -24917.908} C_VEL
LIN {X 0,Y 134.026,Z 543.662,A -85,B 0,C 180,E1 -24918.706,E2 -24918.706} C_VEL
LIN {X 0,Y 132.997,Z 544.917,A -85,B 0,C 180,E1 -24921.152,E2 -24921.152} C_VEL
LIN {X 0,Y 131.231,Z 545.829,A -85,B 0,C 180,E1 -24923.58,E2 -24923.58} C_VEL
LIN {X 0,Y 127.435,Z 546.886,A -85,B 0,C 180,E1 -24928.603,E2 -24928.603} C_VEL
LIN {X 0,Y 126.302,Z 547.05,A -85,B 0,C 180,E1 -24932.172,E2 -24932.172} C_VEL
LIN {X 0,Y 126.391,Z 546.768,A -85,B 0,C 180,E1 -24936.385,E2 -24936.385} C_VEL
LIN {X 0,Y 127.263,Z 545.086,A -85,B 0,C 180,E1 -24942.762,E2 -24942.762} C_VEL
LIN {X 0,Y 129.406,Z 541.942,A -85,B 0,C 180,E1 -24949.017,E2 -24949.017} C_VEL
LIN {X 0,Y 131.915,Z 538.512,A -85,B 0,C 180,E1 -24953.551,E2 -24953.551} C_VEL
LIN {X 0,Y 135.081,Z 534.141,A -85,B 0,C 180,E1 -24957.92,E2 -24957.92} C_VEL
LIN {X 0,Y 139.737,Z 527.707,A -85,B 0,C 180,E1 -24962.728,E2 -24962.728} C_VEL
LIN {X 0,Y 145.366,Z 519.625,A -85,B 0,C 180,E1 -24967.18,E2 -24967.18} C_VEL
LIN {X 0,Y 150.906,Z 511.054,A -85,B 0,C 180,E1 -24970.692,E2 -24970.692} C_VEL
LIN {X 0,Y 156.414,Z 501.435,A -85,B 0,C 180,E1 -24973.726,E2 -24973.726} C_VEL
LIN {X 0,Y 161.648,Z 490.972,A -85,B 0,C 180,E1 -24976.286,E2 -24976.286} C_VEL
LIN {X 0,Y 166.721,Z 479.374,A -85,B 0,C 180,E1 -24978.437,E2 -24978.437} C_VEL
LIN {X 0,Y 171.442,Z 466.463,A -85,B 0,C 180,E1 -24980.23,E2 -24980.23} C_VEL
LIN {X 0,Y 175.085,Z 453.936,A -85,B 0,C 180,E1 -24981.511,E2 -24981.511} C_VEL
LIN {X 0,Y 178.078,Z 440.387,A -85,B 0,C 180,E1 -24982.466,E2 -24982.466} C_VEL
LIN {X 0,Y 180.075,Z 425.998,A -85,B 0,C 180,E1 -24983.147,E2 -24983.147} C_VEL
LIN {X 0,Y 184.073,Z 376.824,A -85,B 0,C 180,E1 -24984.747,E2 -24984.747} C_VEL
LIN {X 0,Y 180.299,Z 368.005,A -85,B 0,C 180,E1 -24987.093,E2 -24987.093} C_VEL
LIN {X 0,Y 175.373,Z 358.027,A -85,B 0,C 180,E1 -24990.435,E2 -24990.435} C_VEL
LIN {X 0,Y 170.778,Z 349.794,A -85,B 0,C 180,E1 -24993.99,E2 -24993.99} C_VEL
LIN {X 0,Y 168.017,Z 345.269,A -85,B 0,C 180,E1 -24996.423,E2 -24996.423} C_VEL
LIN {X 0,Y 165.431,Z 341.248,A -85,B 0,C 180,E1 -24998.996,E2 -24998.996} C_VEL
LIN {X 0,Y 162.18,Z 336.51,A -85,B 0,C 180,E1 -25002.83,E2 -25002.83} C_VEL
LIN {X 0,Y 158.657,Z 331.48,A -85,B 0,C 180,E1 -25008.503,E2 -25008.503} C_VEL
LIN {X 0,Y 156.684,Z 328.991,A -85,B 0,C 180,E1 -25013.562,E2 -25013.562} C_VEL
LIN {X 0,Y 155.786,Z 327.442,A -85,B 0,C 180,E1 -25020.001,E2 -25020.001} C_VEL
LIN {X 0,Y 156.681,Z 329.469,A -85,B 0,C 180,E1 -25027.248,E2 -25027.248} C_VEL
LIN {X 0,Y 159.635,Z 333.872,A -85,B 0,C 180,E1 -25034.176,E2 -25034.176} C_VEL
LIN {X 0,Y 163.618,Z 340.047,A -85,B 0,C 180,E1 -25039.828,E2 -25039.828} C_VEL
LIN {X 0,Y 166.942,Z 345.427,A -85,B 0,C 180,E1 -25043.416,E2 -25043.416} C_VEL
LIN {X 0,Y 170.217,Z 351.273,A -85,B 0,C 180,E1 -25046.433,E2 -25046.433} C_VEL
LIN {X 0,Y 173.77,Z 357.903,A -85,B 0,C 180,E1 -25049.284,E2 -25049.284} C_VEL
LIN {X 0,Y 178.721,Z 368.323,A -85,B 0,C 180,E1 -25052.78,E2 -25052.78} C_VEL
LIN {X 0,Y 182.898,Z 378.503,A -85,B 0,C 180,E1 -25055.451,E2 -25055.451} C_VEL
LIN {X 0,Y 183.651,Z 380.475,A -85,B 0,C 180,E1 -25055.91,E2 -25055.91} C_VEL
LIN {X 0,Y 179.821,Z 428.498,A -85,B 0,C 180,E1 -25057.435,E2 -25057.435} C_VEL
LIN {X 0,Y 177.654,Z 442.095,A -85,B 0,C 180,E1 -25058.164,E2 -25058.164} C_VEL
LIN {X 0,Y 174.575,Z 455.097,A -85,B 0,C 180,E1 -25059.199,E2 -25059.199} C_VEL
LIN {X 0,Y 171.082,Z 466.766,A -85,B 0,C 180,E1 -25060.539,E2 -25060.539} C_VEL
LIN {X 0,Y 166.512,Z 479.007,A -85,B 0,C 180,E1 -25062.412,E2 -25062.412} C_VEL
LIN {X 0,Y 161.632,Z 489.797,A -85,B 0,C 180,E1 -25064.602,E2 -25064.602} C_VEL
LIN {X 0,Y 155.792,Z 500.547,A -85,B 0,C 180,E1 -25067.417,E2 -25067.417} C_VEL
LIN {X 0,Y 149.945,Z 510.052,A -85,B 0,C 180,E1 -25070.747,E2 -25070.747} C_VEL
LIN {X 0,Y 144.641,Z 517.753,A -85,B 0,C 180,E1 -25074.334,E2 -25074.334} C_VEL
LIN {X 0,Y 139.949,Z 524.019,A -85,B 0,C 180,E1 -25078.178,E2 -25078.178} C_VEL
LIN {X 0,Y 135.989,Z 529.078,A -85,B 0,C 180,E1 -25082.282,E2 -25082.282} C_VEL
LIN {X 0,Y 132.69,Z 533.061,A -85,B 0,C 180,E1 -25086.594,E2 -25086.594} C_VEL
LIN {X 0,Y 130.007,Z 536.086,A -85,B 0,C 180,E1 -25091.074,E2 -25091.074} C_VEL
LIN {X 0,Y 127.75,Z 538.776,A -85,B 0,C 180,E1 -25097.288,E2 -25097.288} C_VEL
LIN {X 0,Y 126.586,Z 539.945,A -85,B 0,C 180,E1 -25103.625,E2 -25103.625} C_VEL
LIN {X 0,Y 126.447,Z 539.99,A -85,B 0,C 180,E1 -25106.814,E2 -25106.814} C_VEL
LIN {X 0,Y 126.476,Z 539.684,A -85,B 0,C 180,E1 -25110,E2 -25110} C_VEL
LIN {X 0,Y 127.171,Z 538.014,A -85,B 0,C 180,E1 -25116.345,E2 -25116.345} C_VEL
LIN {X 0,Y 127.889,Z 536.631,A -85,B 0,C 180,E1 -25119.489,E2 -25119.489} C_VEL
LIN {X 0,Y 129.56,Z 533.79,A -85,B 0,C 180,E1 -25124.128,E2 -25124.128} C_VEL
LIN {X 0,Y 131.867,Z 530.022,A -85,B 0,C 180,E1 -25128.649,E2 -25128.649} C_VEL
LIN {X 0,Y 134.988,Z 525.229,A -85,B 0,C 180,E1 -25132.984,E2 -25132.984} C_VEL
LIN {X 0,Y 139.445,Z 518.18,A -85,B 0,C 180,E1 -25137.787,E2 -25137.787} C_VEL
LIN {X 0,Y 143.902,Z 510.644,A -85,B 0,C 180,E1 -25141.668,E2 -25141.668} C_VEL
LIN {X 0,Y 149.035,Z 501.343,A -85,B 0,C 180,E1 -25145.286,E2 -25145.286} C_VEL
LIN {X 0,Y 153.758,Z 491.869,A -85,B 0,C 180,E1 -25148.101,E2 -25148.101} C_VEL
LIN {X 0,Y 158.14,Z 481.501,A -85,B 0,C 180,E1 -25150.537,E2 -25150.537} C_VEL
LIN {X 0,Y 162.554,Z 469.655,A -85,B 0,C 180,E1 -25152.618,E2 -25152.618} C_VEL
LIN {X 0,Y 166.202,Z 457.455,A -85,B 0,C 180,E1 -25154.243,E2 -25154.243} C_VEL
LIN {X 0,Y 169.188,Z 444.146,A -85,B 0,C 180,E1 -25155.526,E2 -25155.526} C_VEL
LIN {X 0,Y 171.373,Z 430.417,A -85,B 0,C 180,E1 -25156.383,E2 -25156.383} C_VEL
LIN {X 0,Y 173.158,Z 409.334,A -85,B 0,C 180,E1 -25157.146,E2 -25157.146} C_VEL
LIN {X 0,Y 175.67,Z 374.374,A -85,B 0,C 180,E1 -25158.307,E2 -25158.307} C_VEL
LIN {X 0,Y 175.344,Z 371.817,A -85,B 0,C 180,E1 -25158.595,E2 -25158.595} C_VEL
LIN {X 0,Y 170.843,Z 360.599,A -85,B 0,C 180,E1 -25161.25,E2 -25161.25} C_VEL
LIN {X 0,Y 165.856,Z 350.075,A -85,B 0,C 180,E1 -25164.454,E2 -25164.454} C_VEL
LIN {X 0,Y 160.701,Z 340.632,A -85,B 0,C 180,E1 -25168.198,E2 -25168.198} C_VEL
LIN {X 0,Y 157.731,Z 335.597,A -85,B 0,C 180,E1 -25170.65,E2 -25170.65} C_VEL
LIN {X 0,Y 154.759,Z 330.952,A -85,B 0,C 180,E1 -25173.395,E2 -25173.395} C_VEL
LIN {X 0,Y 151.032,Z 325.433,A -85,B 0,C 180,E1 -25177.472,E2 -25177.472} C_VEL
LIN {X 0,Y 146.739,Z 319.39,A -85,B 0,C 180,E1 -25183.835,E2 -25183.835} C_VEL
LIN {X 0,Y 143.758,Z 315.624,A -85,B 0,C 180,E1 -25191.565,E2 -25191.565} C_VEL
LIN {X 0,Y 143.127,Z 314.094,A -85,B 0,C 180,E1 -25197.185,E2 -25197.185} C_VEL
LIN {X 0,Y 143.291,Z 313.936,A -85,B 0,C 180,E1 -25200.35,E2 -25200.35} C_VEL
LIN {X 0,Y 146.236,Z 317.761,A -85,B 0,C 180,E1 -25210.382,E2 -25210.382} C_VEL
LIN {X 0,Y 147.402,Z 319.374,A -85,B 0,C 180,E1 -25212.563,E2 -25212.563} C_VEL
LIN {X 0,Y 151.478,Z 324.61,A -85,B 0,C 180,E1 -25218.264,E2 -25218.264} C_VEL
LIN {X 0,Y 155.457,Z 330.138,A -85,B 0,C 180,E1 -25222.477,E2 -25222.477} C_VEL
LIN {X 0,Y 158.914,Z 335.458,A -85,B 0,C 180,E1 -25225.563,E2 -25225.563} C_VEL
LIN {X 0,Y 162.355,Z 341.021,A -85,B 0,C 180,E1 -25228.258,E2 -25228.258} C_VEL
LIN {X 0,Y 165.961,Z 347.36,A -85,B 0,C 180,E1 -25230.803,E2 -25230.803} C_VEL
LIN {X 0,Y 170.175,Z 355.58,A -85,B 0,C 180,E1 -25233.518,E2 -25233.518} C_VEL
LIN {X 0,Y 174.606,Z 365.413,A -85,B 0,C 180,E1 -25236.151,E2 -25236.151} C_VEL
LIN {X 0,Y 176.267,Z 369.889,A -85,B 0,C 180,E1 -25237.117,E2 -25237.117} C_VEL
LIN {X 0,Y 171.46,Z 430.163,A -85,B 0,C 180,E1 -25239.201,E2 -25239.201} C_VEL
LIN {X 0,Y 169.445,Z 443.636,A -85,B 0,C 180,E1 -25240.004,E2 -25240.004} C_VEL
LIN {X 0,Y 166.284,Z 457.385,A -85,B 0,C 180,E1 -25241.164,E2 -25241.164} C_VEL
LIN {X 0,Y 163.259,Z 468.33,A -85,B 0,C 180,E1 -25242.508,E2 -25242.508} C_VEL
LIN {X 0,Y 158.858,Z 480.938,A -85,B 0,C 180,E1 -25244.49,E2 -25244.49} C_VEL
LIN {X 0,Y 154.306,Z 492.333,A -85,B 0,C 180,E1 -25246.908,E2 -25246.908} C_VEL
LIN {X 0,Y 149.448,Z 502.666,A -85,B 0,C 180,E1 -25249.714,E2 -25249.714} C_VEL
LIN {X 0,Y 144.02,Z 512.778,A -85,B 0,C 180,E1 -25253.29,E2 -25253.29} C_VEL
LIN {X 0,Y 139.355,Z 521.087,A -85,B 0,C 180,E1 -25257.171,E2 -25257.171} C_VEL
LIN {X 0,Y 134.809,Z 528.952,A -85,B 0,C 180,E1 -25262.019,E2 -25262.019} C_VEL
LIN {X 0,Y 131.753,Z 534.361,A -85,B 0,C 180,E1 -25266.418,E2 -25266.418} C_VEL
LIN {X 0,Y 129.298,Z 538.706,A -85,B 0,C 180,E1 -25270.966,E2 -25270.966} C_VEL
LIN {X 0,Y 127.212,Z 543.015,A -85,B 0,C 180,E1 -25277.234,E2 -25277.234} C_VEL
LIN {X 0,Y 126.364,Z 545.776,A -85,B 0,C 180,E1 -25283.614,E2 -25283.614} C_VEL
LIN {X 0,Y 126.299,Z 546.578,A -85,B 0,C 180,E1 -25286.81,E2 -25286.81} C_VEL
LIN {X 0,Y 126.426,Z 547.01,A -85,B 0,C 180,E1 -25290,E2 -25290} C_VEL
LIN {X 0,Y 126.302,Z 547.05,A -85,B 0,C 180,E1 -25292.172,E2 -25292.172} C_VEL
LIN {X 0,Y 125.983,Z 547.018,A -85,B 0,C 180,E1 -25293.951,E2 -25293.951} C_VEL
LIN {X 0,Y 124.73,Z 546.723,A -85,B 0,C 180,E1 -25296.593,E2 -25296.593} C_VEL
LIN {X 0,Y 121.254,Z 545.121,A -85,B 0,C 180,E1 -25302.853,E2 -25302.853} C_VEL
LIN {X 0,Y 120.933,Z 544.069,A -85,B 0,C 180,E1 -25305.627,E2 -25305.627} C_VEL
LIN {X 0,Y 121.149,Z 543.649,A -85,B 0,C 180,E1 -25306.546,E2 -25306.546} C_VEL
LIN {X 0,Y 123.522,Z 540.717,A -85,B 0,C 180,E1 -25311.705,E2 -25311.705} C_VEL
LIN {X 0,Y 126.49,Z 537.017,A -85,B 0,C 180,E1 -25316.391,E2 -25316.391} C_VEL
LIN {X 0,Y 130.126,Z 532.339,A -85,B 0,C 180,E1 -25320.869,E2 -25320.869} C_VEL
LIN {X 0,Y 135.401,Z 525.442,A -85,B 0,C 180,E1 -25325.727,E2 -25325.727} C_VEL
LIN {X 0,Y 140.654,Z 518.154,A -85,B 0,C 180,E1 -25329.573,E2 -25329.573} C_VEL
LIN {X 0,Y 146.623,Z 509.292,A -85,B 0,C 180,E1 -25333.081,E2 -25333.081} C_VEL
LIN {X 0,Y 152.174,Z 499.802,A -85,B 0,C 180,E1 -25336.003,E2 -25336.003} C_VEL
LIN {X 0,Y 157.981,Z 488.502,A -85,B 0,C 180,E1 -25338.651,E2 -25338.651} C_VEL
LIN {X 0,Y 163.29,Z 476.363,A -85,B 0,C 180,E1 -25340.779,E2 -25340.779} C_VEL
LIN {X 0,Y 167.599,Z 464.466,A -85,B 0,C 180,E1 -25342.324,E2 -25342.324} C_VEL
LIN {X 0,Y 171.397,Z 451.243,A -85,B 0,C 180,E1 -25343.581,E2 -25343.581} C_VEL
LIN {X 0,Y 174.238,Z 438.035,A -85,B 0,C 180,E1 -25344.441,E2 -25344.441} C_VEL
LIN {X 0,Y 176.097,Z 423.96,A -85,B 0,C 180,E1 -25345.062,E2 -25345.062} C_VEL
LIN {X 0,Y 179.82,Z 379.56,A -85,B 0,C 180,E1 -25346.493,E2 -25346.493} C_VEL
LIN {X 0,Y 175.757,Z 370.024,A -85,B 0,C 180,E1 -25349.265,E2 -25349.265} C_VEL
LIN {X 0,Y 171.186,Z 360.754,A -85,B 0,C 180,E1 -25352.725,E2 -25352.725} C_VEL
LIN {X 0,Y 167.629,Z 354.319,A -85,B 0,C 180,E1 -25355.79,E2 -25355.79} C_VEL
LIN {X 0,Y 165.636,Z 350.953,A -85,B 0,C 180,E1 -25357.715,E2 -25357.715} C_VEL
LIN {X 0,Y 163.601,Z 347.609,A -85,B 0,C 180,E1 -25359.9,E2 -25359.9} C_VEL
LIN {X 0,Y 160.742,Z 343.211,A -85,B 0,C 180,E1 -25363.49,E2 -25363.49} C_VEL
LIN {X 0,Y 157.455,Z 338.25,A -85,B 0,C 180,E1 -25369.13,E2 -25369.13} C_VEL
LIN {X 0,Y 155.644,Z 335.895,A -85,B 0,C 180,E1 -25374.17,E2 -25374.17} C_VEL
LIN {X 0,Y 154.919,Z 334.5,A -85,B 0,C 180,E1 -25380.001,E2 -25380.001} C_VEL
LIN {X 0,Y 155.75,Z 336.47,A -85,B 0,C 180,E1 -25387.048,E2 -25387.048} C_VEL
LIN {X 0,Y 158.248,Z 340.423,A -85,B 0,C 180,E1 -25393.321,E2 -25393.321} C_VEL
LIN {X 0,Y 161.87,Z 346.41,A -85,B 0,C 180,E1 -25398.881,E2 -25398.881} C_VEL
LIN {X 0,Y 164.964,Z 351.726,A -85,B 0,C 180,E1 -25402.465,E2 -25402.465} C_VEL
LIN {X 0,Y 167.673,Z 356.722,A -85,B 0,C 180,E1 -25405.144,E2 -25405.144} C_VEL
LIN {X 0,Y 170.965,Z 363.165,A -85,B 0,C 180,E1 -25407.993,E2 -25407.993} C_VEL
LIN {X 0,Y 175.737,Z 373.699,A -85,B 0,C 180,E1 -25411.626,E2 -25411.626} C_VEL
LIN {X 0,Y 179.376,Z 383.065,A -85,B 0,C 180,E1 -25414.136,E2 -25414.136} C_VEL
LIN {X 0,Y 175.636,Z 428.468,A -85,B 0,C 180,E1 -25415.595,E2 -25415.595} C_VEL
LIN {X 0,Y 173.362,Z 442.209,A -85,B 0,C 180,E1 -25416.321,E2 -25416.321} C_VEL
LIN {X 0,Y 170.187,Z 455.198,A -85,B 0,C 180,E1 -25417.351,E2 -25417.351} C_VEL
LIN {X 0,Y 166.549,Z 466.863,A -85,B 0,C 180,E1 -25418.68,E2 -25418.68} C_VEL
LIN {X 0,Y 162.236,Z 478.039,A -85,B 0,C 180,E1 -25420.364,E2 -25420.364} C_VEL
LIN {X 0,Y 157.287,Z 488.828,A -85,B 0,C 180,E1 -25422.502,E2 -25422.502} C_VEL
LIN {X 0,Y 151.739,Z 498.887,A -85,B 0,C 180,E1 -25425.064,E2 -25425.064} C_VEL
LIN {X 0,Y 146.445,Z 507.225,A -85,B 0,C 180,E1 -25427.789,E2 -25427.789} C_VEL
LIN {X 0,Y 140.712,Z 515.46,A -85,B 0,C 180,E1 -25431.368,E2 -25431.368} C_VEL
LIN {X 0,Y 135.49,Z 522.184,A -85,B 0,C 180,E1 -25435.21,E2 -25435.21} C_VEL
LIN {X 0,Y 131.197,Z 527.483,A -85,B 0,C 180,E1 -25439.236,E2 -25439.236} C_VEL
LIN {X 0,Y 127.325,Z 531.996,A -85,B 0,C 180,E1 -25443.796,E2 -25443.796} C_VEL
LIN {X 0,Y 123.279,Z 536.256,A -85,B 0,C 180,E1 -25449.998,E2 -25449.998} C_VEL
LIN {X 0,Y 120.81,Z 538.956,A -85,B 0,C 180,E1 -25456.544,E2 -25456.544} C_VEL
LIN {X 0,Y 119.542,Z 540.141,A -85,B 0,C 180,E1 -25463.247,E2 -25463.247} C_VEL
LIN {X 0,Y 119.363,Z 540.192,A -85,B 0,C 180,E1 -25466.624,E2 -25466.624} C_VEL
LIN {X 0,Y 119.396,Z 539.891,A -85,B 0,C 180,E1 -25470,E2 -25470} C_VEL
LIN {X 0,Y 120.119,Z 538.233,A -85,B 0,C 180,E1 -25476.72,E2 -25476.72} C_VEL
LIN {X 0,Y 120.912,Z 536.859,A -85,B 0,C 180,E1 -25480.042,E2 -25480.042} C_VEL
LIN {X 0,Y 122.698,Z 534.028,A -85,B 0,C 180,E1 -25484.936,E2 -25484.936} C_VEL
LIN {X 0,Y 125.178,Z 530.275,A -85,B 0,C 180,E1 -25489.685,E2 -25489.685} C_VEL
LIN {X 0,Y 128.48,Z 525.501,A -85,B 0,C 180,E1 -25494.22,E2 -25494.22} C_VEL
LIN {X 0,Y 133.223,Z 518.471,A -85,B 0,C 180,E1 -25499.206,E2 -25499.206} C_VEL
LIN {X 0,Y 137.919,Z 510.961,A -85,B 0,C 180,E1 -25503.215,E2 -25503.215} C_VEL
LIN {X 0,Y 143.323,Z 501.708,A -85,B 0,C 180,E1 -25506.918,E2 -25506.918} C_VEL
LIN {X 0,Y 148.256,Z 492.278,A -85,B 0,C 180,E1 -25509.788,E2 -25509.788} C_VEL
LIN {X 0,Y 152.828,Z 481.969,A -85,B 0,C 180,E1 -25512.263,E2 -25512.263} C_VEL
LIN {X 0,Y 157.058,Z 471.219,A -85,B 0,C 180,E1 -25514.202,E2 -25514.202} C_VEL
LIN {X 0,Y 160.639,Z 460.1,A -85,B 0,C 180,E1 -25515.758,E2 -25515.758} C_VEL
LIN {X 0,Y 163.747,Z 447.683,A -85,B 0,C 180,E1 -25517.068,E2 -25517.068} C_VEL
LIN {X 0,Y 166.306,Z 434.092,A -85,B 0,C 180,E1 -25518.019,E2 -25518.019} C_VEL
LIN {X 0,Y 167.808,Z 420.38,A -85,B 0,C 180,E1 -25518.604,E2 -25518.604} C_VEL
LIN {X 0,Y 171.202,Z 375.512,A -85,B 0,C 180,E1 -25520.086,E2 -25520.086} C_VEL
LIN {X 0,Y 167.225,Z 365.16,A -85,B 0,C 180,E1 -25522.631,E2 -25522.631} C_VEL
LIN {X 0,Y 162.733,Z 355.23,A -85,B 0,C 180,E1 -25525.75,E2 -25525.75} C_VEL
LIN {X 0,Y 157.677,Z 345.632,A -85,B 0,C 180,E1 -25529.728,E2 -25529.728} C_VEL
LIN {X 0,Y 155.034,Z 341.029,A -85,B 0,C 180,E1 -25532.105,E2 -25532.105} C_VEL
LIN {X 0,Y 152.706,Z 337.169,A -85,B 0,C 180,E1 -25534.438,E2 -25534.438} C_VEL
LIN {X 0,Y 149.4,Z 331.982,A -85,B 0,C 180,E1 -25538.313,E2 -25538.313} C_VEL
LIN {X 0,Y 145.356,Z 326.01,A -85,B 0,C 180,E1 -25544.756,E2 -25544.756} C_VEL
LIN {X 0,Y 142.686,Z 322.32,A -85,B 0,C 180,E1 -25552.57,E2 -25552.57} C_VEL
LIN {X 0,Y 142.298,Z 320.928,A -85,B 0,C 180,E1 -25558.584,E2 -25558.584} C_VEL
LIN {X 0,Y 142.45,Z 321.131,A -85,B 0,C 180,E1 -25560.706,E2 -25560.706} C_VEL
LIN {X 0,Y 145.194,Z 324.761,A -85,B 0,C 180,E1 -25570.105,E2 -25570.105} C_VEL
LIN {X 0,Y 149.76,Z 331.091,A -85,B 0,C 180,E1 -25577.364,E2 -25577.364} C_VEL
LIN {X 0,Y 153.411,Z 336.452,A -85,B 0,C 180,E1 -25581.499,E2 -25581.499} C_VEL
LIN {X 0,Y 156.49,Z 341.395,A -85,B 0,C 180,E1 -25584.438,E2 -25584.438} C_VEL
LIN {X 0,Y 159.467,Z 346.377,A -85,B 0,C 180,E1 -25586.943,E2 -25586.943} C_VEL
LIN {X 0,Y 163.59,Z 354.003,A -85,B 0,C 180,E1 -25590.05,E2 -25590.05} C_VEL
LIN {X 0,Y 167.65,Z 362.422,A -85,B 0,C 180,E1 -25592.821,E2 -25592.821} C_VEL
LIN {X 0,Y 171.636,Z 371.989,A -85,B 0,C 180,E1 -25595.335,E2 -25595.335} C_VEL
LIN {X 0,Y 166.903,Z 429.905,A -85,B 0,C 180,E1 -25597.366,E2 -25597.366} C_VEL
LIN {X 0,Y 164.808,Z 443.447,A -85,B 0,C 180,E1 -25598.166,E2 -25598.166} C_VEL
LIN {X 0,Y 161.383,Z 457.792,A -85,B 0,C 180,E1 -25599.378,E2 -25599.378} C_VEL
LIN {X 0,Y 157.939,Z 469.516,A -85,B 0,C 180,E1 -25600.848,E2 -25600.848} C_VEL
LIN {X 0,Y 153.379,Z 481.878,A -85,B 0,C 180,E1 -25602.851,E2 -25602.851} C_VEL
LIN {X 0,Y 148.595,Z 493.172,A -85,B 0,C 180,E1 -25605.345,E2 -25605.345} C_VEL
LIN {X 0,Y 143.099,Z 504.108,A -85,B 0,C 180,E1 -25608.47,E2 -25608.47} C_VEL
LIN {X 0,Y 137.456,Z 513.952,A -85,B 0,C 180,E1 -25612.154,E2 -25612.154} C_VEL
LIN {X 0,Y 132.626,Z 522.032,A -85,B 0,C 180,E1 -25616.193,E2 -25616.193} C_VEL
LIN {X 0,Y 128.512,Z 528.67,A -85,B 0,C 180,E1 -25620.516,E2 -25620.516} C_VEL
LIN {X 0,Y 125.229,Z 534.099,A -85,B 0,C 180,E1 -25625.109,E2 -25625.109} C_VEL
LIN {X 0,Y 122.551,Z 538.46,A -85,B 0,C 180,E1 -25629.875,E2 -25629.875} C_VEL
LIN {X 0,Y 120.235,Z 542.782,A -85,B 0,C 180,E1 -25636.479,E2 -25636.479} C_VEL
LIN {X 0,Y 119.278,Z 545.558,A -85,B 0,C 180,E1 -25643.233,E2 -25643.233} C_VEL
LIN {X 0,Y 119.193,Z 546.371,A -85,B 0,C 180,E1 -25646.62,E2 -25646.62} C_VEL
LIN {X 0,Y 119.331,Z 546.809,A -85,B 0,C 180,E1 -25650,E2 -25650} C_VEL
LIN {X 0,Y 119.219,Z 546.872,A -85,B 0,C 180,E1 -25653.38,E2 -25653.38} C_VEL
LIN {X 0,Y 119.641,Z 545.92,A -85,B 0,C 180,E1 -25660.15,E2 -25660.15} C_VEL
LIN {X 0,Y 121.149,Z 543.649,A -85,B 0,C 180,E1 -25666.546,E2 -25666.546} C_VEL
LIN {X 0,Y 121.534,Z 542.39,A -85,B 0,C 180,E1 -25669.271,E2 -25669.271} C_VEL
LIN {X 0,Y 120.927,Z 539.791,A -85,B 0,C 180,E1 -25673.797,E2 -25673.797} C_VEL
LIN {X 0,Y 120.79,Z 537.224,A -85,B 0,C 180,E1 -25677.376,E2 -25677.376} C_VEL
LIN {X 0,Y 121.723,Z 534.995,A -85,B 0,C 180,E1 -25679.934,E2 -25679.934} C_VEL
LIN {X 0,Y 122.332,Z 534.174,A -85,B 0,C 180,E1 -25680.732,E2 -25680.732} C_VEL
LIN {X 0,Y 127.961,Z 527.42,A -85,B 0,C 180,E1 -25686.186,E2 -25686.186} C_VEL
LIN {X 0,Y 134.255,Z 519.356,A -85,B 0,C 180,E1 -25690.87,E2 -25690.87} C_VEL
LIN {X 0,Y 140.431,Z 510.805,A -85,B 0,C 180,E1 -25694.478,E2 -25694.478} C_VEL
LIN {X 0,Y 146.892,Z 500.417,A -85,B 0,C 180,E1 -25697.798,E2 -25697.798} C_VEL
LIN {X 0,Y 152.758,Z 489.567,A -85,B 0,C 180,E1 -25700.409,E2 -25700.409} C_VEL
LIN {X 0,Y 158.275,Z 477.723,A -85,B 0,C 180,E1 -25702.533,E2 -25702.533} C_VEL
LIN {X 0,Y 162.714,Z 466.238,A -85,B 0,C 180,E1 -25704.081,E2 -25704.081} C_VEL
LIN {X 0,Y 166.627,Z 453.691,A -85,B 0,C 180,E1 -25705.332,E2 -25705.332} C_VEL
LIN {X 0,Y 169.783,Z 440.168,A -85,B 0,C 180,E1 -25706.264,E2 -25706.264} C_VEL
LIN {X 0,Y 171.834,Z 426.527,A -85,B 0,C 180,E1 -25706.899,E2 -25706.899} C_VEL
LIN {X 0,Y 175.706,Z 382.337,A -85,B 0,C 180,E1 -25708.334,E2 -25708.334} C_VEL
LIN {X 0,Y 171.722,Z 372.957,A -85,B 0,C 180,E1 -25711.322,E2 -25711.322} C_VEL
LIN {X 0,Y 167.695,Z 364.548,A -85,B 0,C 180,E1 -25714.727,E2 -25714.727} C_VEL
LIN {X 0,Y 163.887,Z 357.533,A -85,B 0,C 180,E1 -25718.459,E2 -25718.459} C_VEL
LIN {X 0,Y 161.689,Z 353.78,A -85,B 0,C 180,E1 -25720.975,E2 -25720.975} C_VEL
LIN {X 0,Y 159.013,Z 349.501,A -85,B 0,C 180,E1 -25724.623,E2 -25724.623} C_VEL
LIN {X 0,Y 156.206,Z 344.968,A -85,B 0,C 180,E1 -25729.913,E2 -25729.913} C_VEL
LIN {X 0,Y 154.624,Z 342.778,A -85,B 0,C 180,E1 -25734.785,E2 -25734.785} C_VEL
LIN {X 0,Y 154.054,Z 341.55,A -85,B 0,C 180,E1 -25740.001,E2 -25740.001} C_VEL
LIN {X 0,Y 154.815,Z 343.515,A -85,B 0,C 180,E1 -25746.845,E2 -25746.845} C_VEL
LIN {X 0,Y 157.038,Z 347.316,A -85,B 0,C 180,E1 -25752.767,E2 -25752.767} C_VEL
LIN {X 0,Y 160.232,Z 352.878,A -85,B 0,C 180,E1 -25758.001,E2 -25758.001} C_VEL
LIN {X 0,Y 162.99,Z 357.893,A -85,B 0,C 180,E1 -25761.437,E2 -25761.437} C_VEL
LIN {X 0,Y 165.904,Z 363.56,A -85,B 0,C 180,E1 -25764.491,E2 -25764.491} C_VEL
LIN {X 0,Y 169.251,Z 370.782,A -85,B 0,C 180,E1 -25767.552,E2 -25767.552} C_VEL
LIN {X 0,Y 172.858,Z 379.211,A -85,B 0,C 180,E1 -25770.462,E2 -25770.462} C_VEL
LIN {X 0,Y 175.321,Z 385.855,A -85,B 0,C 180,E1 -25772.312,E2 -25772.312} C_VEL
LIN {X 0,Y 171.591,Z 428.731,A -85,B 0,C 180,E1 -25773.675,E2 -25773.675} C_VEL
LIN {X 0,Y 169.252,Z 442.323,A -85,B 0,C 180,E1 -25774.384,E2 -25774.384} C_VEL
LIN {X 0,Y 165.985,Z 455.299,A -85,B 0,C 180,E1 -25775.407,E2 -25775.407} C_VEL
LIN {X 0,Y 162.215,Z 466.96,A -85,B 0,C 180,E1 -25776.726,E2 -25776.726} C_VEL
LIN {X 0,Y 157.301,Z 479.138,A -85,B 0,C 180,E1 -25778.571,E2 -25778.571} C_VEL
LIN {X 0,Y 152,Z 490.008,A -85,B 0,C 180,E1 -25780.789,E2 -25780.789} C_VEL
LIN {X 0,Y 145.645,Z 500.772,A -85,B 0,C 180,E1 -25783.63,E2 -25783.63} C_VEL
LIN {X 0,Y 139.218,Z 510.295,A -85,B 0,C 180,E1 -25787.039,E2 -25787.039} C_VEL
LIN {X 0,Y 133.334,Z 518.018,A -85,B 0,C 180,E1 -25790.765,E2 -25790.765} C_VEL
LIN {X 0,Y 128.038,Z 524.304,A -85,B 0,C 180,E1 -25794.807,E2 -25794.807} C_VEL
LIN {X 0,Y 123.557,Z 529.378,A -85,B 0,C 180,E1 -25799.208,E2 -25799.208} C_VEL
LIN {X 0,Y 119.744,Z 533.379,A -85,B 0,C 180,E1 -25803.884,E2 -25803.884} C_VEL
LIN {X 0,Y 116.601,Z 536.426,A -85,B 0,C 180,E1 -25808.799,E2 -25808.799} C_VEL
LIN {X 0,Y 113.901,Z 539.137,A -85,B 0,C 180,E1 -25815.711,E2 -25815.711} C_VEL
LIN {X 0,Y 112.487,Z 540.338,A -85,B 0,C 180,E1 -25822.822,E2 -25822.822} C_VEL
LIN {X 0,Y 112.274,Z 540.393,A -85,B 0,C 180,E1 -25826.411,E2 -25826.411} C_VEL
LIN {X 0,Y 112.307,Z 540.098,A -85,B 0,C 180,E1 -25830,E2 -25830} C_VEL
LIN {X 0,Y 113.085,Z 538.451,A -85,B 0,C 180,E1 -25837.14,E2 -25837.14} C_VEL
LIN {X 0,Y 113.946,Z 537.085,A -85,B 0,C 180,E1 -25840.663,E2 -25840.663} C_VEL
LIN {X 0,Y 115.86,Z 534.266,A -85,B 0,C 180,E1 -25845.84,E2 -25845.84} C_VEL
LIN {X 0,Y 118.519,Z 530.529,A -85,B 0,C 180,E1 -25850.841,E2 -25850.841} C_VEL
LIN {X 0,Y 122.04,Z 525.772,A -85,B 0,C 180,E1 -25855.588,E2 -25855.588} C_VEL
LIN {X 0,Y 127.096,Z 518.762,A -85,B 0,C 180,E1 -25860.763,E2 -25860.763} C_VEL
LIN {X 0,Y 132.053,Z 511.276,A -85,B 0,C 180,E1 -25864.898,E2 -25864.898} C_VEL
LIN {X 0,Y 137.738,Z 502.072,A -85,B 0,C 180,E1 -25868.685,E2 -25868.685} C_VEL
LIN {X 0,Y 142.893,Z 492.686,A -85,B 0,C 180,E1 -25871.603,E2 -25871.603} C_VEL
LIN {X 0,Y 147.666,Z 482.435,A -85,B 0,C 180,E1 -25874.111,E2 -25874.111} C_VEL
LIN {X 0,Y 151.867,Z 472.342,A -85,B 0,C 180,E1 -25875.963,E2 -25875.963} C_VEL
LIN {X 0,Y 155.803,Z 460.759,A -85,B 0,C 180,E1 -25877.615,E2 -25877.615} C_VEL
LIN {X 0,Y 159.32,Z 447.314,A -85,B 0,C 180,E1 -25879.031,E2 -25879.031} C_VEL
LIN {X 0,Y 161.797,Z 434.538,A -85,B 0,C 180,E1 -25879.92,E2 -25879.92} C_VEL
LIN {X 0,Y 163.353,Z 421.158,A -85,B 0,C 180,E1 -25880.51,E2 -25880.51} C_VEL
LIN {X 0,Y 166.693,Z 377.686,A -85,B 0,C 180,E1 -25881.992,E2 -25881.992} C_VEL
LIN {X 0,Y 163.286,Z 368.698,A -85,B 0,C 180,E1 -25884.378,E2 -25884.378} C_VEL
LIN {X 0,Y 159.384,Z 359.855,A -85,B 0,C 180,E1 -25887.332,E2 -25887.332} C_VEL
LIN {X 0,Y 155.318,Z 351.661,A -85,B 0,C 180,E1 -25890.806,E2 -25890.806} C_VEL
LIN {X 0,Y 152.805,Z 347.061,A -85,B 0,C 180,E1 -25893.233,E2 -25893.233} C_VEL
LIN {X 0,Y 150.612,Z 343.266,A -85,B 0,C 180,E1 -25895.602,E2 -25895.602} C_VEL
LIN {X 0,Y 147.679,Z 338.396,A -85,B 0,C 180,E1 -25899.32,E2 -25899.32} C_VEL
LIN {X 0,Y 144.221,Z 332.947,A -85,B 0,C 180,E1 -25905.219,E2 -25905.219} C_VEL
LIN {X 0,Y 141.781,Z 329.367,A -85,B 0,C 180,E1 -25912.737,E2 -25912.737} C_VEL
LIN {X 0,Y 141.43,Z 327.995,A -85,B 0,C 180,E1 -25918.575,E2 -25918.575} C_VEL
LIN {X 0,Y 141.581,Z 328.199,A -85,B 0,C 180,E1 -25920.71,E2 -25920.71} C_VEL
LIN {X 0,Y 144.24,Z 331.829,A -85,B 0,C 180,E1 -25929.995,E2 -25929.995} C_VEL
LIN {X 0,Y 148.144,Z 337.695,A -85,B 0,C 180,E1 -25936.537,E2 -25936.537} C_VEL
LIN {X 0,Y 151.461,Z 342.793,A -85,B 0,C 180,E1 -25940.542,E2 -25940.542} C_VEL
LIN {X 0,Y 154.581,Z 348.113,A -85,B 0,C 180,E1 -25943.707,E2 -25943.707} C_VEL
LIN {X 0,Y 157.97,Z 354.096,A -85,B 0,C 180,E1 -25946.68,E2 -25946.68} C_VEL
LIN {X 0,Y 162.601,Z 363.577,A -85,B 0,C 180,E1 -25950.295,E2 -25950.295} C_VEL
LIN {X 0,Y 166.464,Z 372.774,A -85,B 0,C 180,E1 -25953.017,E2 -25953.017} C_VEL
LIN {X 0,Y 167.176,Z 374.501,A -85,B 0,C 180,E1 -25953.487,E2 -25953.487} C_VEL
LIN {X 0,Y 162.515,Z 429.639,A -85,B 0,C 180,E1 -25955.424,E2 -25955.424} C_VEL
LIN {X 0,Y 160.338,Z 443.253,A -85,B 0,C 180,E1 -25956.218,E2 -25956.218} C_VEL
LIN {X 0,Y 156.974,Z 457.069,A -85,B 0,C 180,E1 -25957.375,E2 -25957.375} C_VEL
LIN {X 0,Y 153.386,Z 468.931,A -85,B 0,C 180,E1 -25958.839,E2 -25958.839} C_VEL
LIN {X 0,Y 148.62,Z 481.383,A -85,B 0,C 180,E1 -25960.835,E2 -25960.835} C_VEL
LIN {X 0,Y 143.583,Z 492.765,A -85,B 0,C 180,E1 -25963.334,E2 -25963.334} C_VEL
LIN {X 0,Y 137.839,Z 503.747,A -85,B 0,C 180,E1 -25966.503,E2 -25966.503} C_VEL
LIN {X 0,Y 131.874,Z 513.623,A -85,B 0,C 180,E1 -25970.245,E2 -25970.245} C_VEL
LIN {X 0,Y 126.736,Z 521.73,A -85,B 0,C 180,E1 -25974.391,E2 -25974.391} C_VEL
LIN {X 0,Y 122.31,Z 528.389,A -85,B 0,C 180,E1 -25978.86,E2 -25978.86} C_VEL
LIN {X 0,Y 118.769,Z 533.836,A -85,B 0,C 180,E1 -25983.654,E2 -25983.654} C_VEL
LIN {X 0,Y 115.862,Z 538.213,A -85,B 0,C 180,E1 -25988.658,E2 -25988.658} C_VEL
LIN {X 0,Y 113.293,Z 542.55,A -85,B 0,C 180,E1 -25995.633,E2 -25995.633} C_VEL
LIN {X 0,Y 112.216,Z 545.341,A -85,B 0,C 180,E1 -26002.805,E2 -26002.805} C_VEL
LIN {X 0,Y 112.107,Z 546.163,A -85,B 0,C 180,E1 -26006.406,E2 -26006.406} C_VEL
LIN {X 0,Y 112.247,Z 546.607,A -85,B 0,C 180,E1 -26010,E2 -26010} C_VEL
LIN {X 0,Y 112.125,Z 546.676,A -85,B 0,C 180,E1 -26013.594,E2 -26013.594} C_VEL
LIN {X 0,Y 112.641,Z 545.734,A -85,B 0,C 180,E1 -26020.788,E2 -26020.788} C_VEL
LIN {X 0,Y 114.43,Z 543.347,A -85,B 0,C 180,E1 -26027.884,E2 -26027.884} C_VEL
LIN {X 0,Y 116.907,Z 540.55,A -85,B 0,C 180,E1 -26033.001,E2 -26033.001} C_VEL
LIN {X 0,Y 120.097,Z 536.859,A -85,B 0,C 180,E1 -26037.914,E2 -26037.914} C_VEL
LIN {X 0,Y 122.332,Z 534.174,A -85,B 0,C 180,E1 -26040.732,E2 -26040.732} C_VEL
LIN {X 0,Y 123.884,Z 531.702,A -85,B 0,C 180,E1 -26043.125,E2 -26043.125} C_VEL
LIN {X 0,Y 125.183,Z 527.375,A -85,B 0,C 180,E1 -26047.196,E2 -26047.196} C_VEL
LIN {X 0,Y 126.911,Z 522.491,A -85,B 0,C 180,E1 -26051.039,E2 -26051.039} C_VEL
LIN {X 0,Y 129.031,Z 519.12,A -85,B 0,C 180,E1 -26052.991,E2 -26052.991} C_VEL
LIN {X 0,Y 135.44,Z 510.68,A -85,B 0,C 180,E1 -26056.59,E2 -26056.59} C_VEL
LIN {X 0,Y 141.761,Z 501.038,A -85,B 0,C 180,E1 -26059.723,E2 -26059.723} C_VEL
LIN {X 0,Y 147.701,Z 490.631,A -85,B 0,C 180,E1 -26062.284,E2 -26062.284} C_VEL
LIN {X 0,Y 153.414,Z 479.041,A -85,B 0,C 180,E1 -26064.403,E2 -26064.403} C_VEL
LIN {X 0,Y 157.988,Z 467.895,A -85,B 0,C 180,E1 -26065.946,E2 -26065.946} C_VEL
LIN {X 0,Y 162.349,Z 454.717,A -85,B 0,C 180,E1 -26067.291,E2 -26067.291} C_VEL
LIN {X 0,Y 165.74,Z 441.109,A -85,B 0,C 180,E1 -26068.244,E2 -26068.244} C_VEL
LIN {X 0,Y 167.832,Z 428.13,A -85,B 0,C 180,E1 -26068.878,E2 -26068.878} C_VEL
LIN {X 0,Y 171.795,Z 385.79,A -85,B 0,C 180,E1 -26070.198,E2 -26070.198} C_VEL
LIN {X 0,Y 171.342,Z 384.127,A -85,B 0,C 180,E1 -26070.599,E2 -26070.599} C_VEL
LIN {X 0,Y 167.416,Z 374.806,A -85,B 0,C 180,E1 -26073.929,E2 -26073.929} C_VEL
LIN {X 0,Y 163.781,Z 367.227,A -85,B 0,C 180,E1 -26077.449,E2 -26077.449} C_VEL
LIN {X 0,Y 161.518,Z 363.002,A -85,B 0,C 180,E1 -26079.959,E2 -26079.959} C_VEL
LIN {X 0,Y 159.835,Z 359.96,A -85,B 0,C 180,E1 -26082.075,E2 -26082.075} C_VEL
LIN {X 0,Y 157.636,Z 356.2,A -85,B 0,C 180,E1 -26085.312,E2 -26085.312} C_VEL
LIN {X 0,Y 155.108,Z 351.854,A -85,B 0,C 180,E1 -26090.403,E2 -26090.403} C_VEL
LIN {X 0,Y 153.759,Z 349.852,A -85,B 0,C 180,E1 -26094.756,E2 -26094.756} C_VEL
LIN {X 0,Y 153.187,Z 348.61,A -85,B 0,C 180,E1 -26100.001,E2 -26100.001} C_VEL
LIN {X 0,Y 153.863,Z 350.519,A -85,B 0,C 180,E1 -26106.558,E2 -26106.558} C_VEL
LIN {X 0,Y 155.807,Z 354.121,A -85,B 0,C 180,E1 -26112.125,E2 -26112.125} C_VEL
LIN {X 0,Y 158.662,Z 359.387,A -85,B 0,C 180,E1 -26117.149,E2 -26117.149} C_VEL
LIN {X 0,Y 161.291,Z 364.497,A -85,B 0,C 180,E1 -26120.652,E2 -26120.652} C_VEL
LIN {X 0,Y 164.246,Z 370.579,A -85,B 0,C 180,E1 -26123.918,E2 -26123.918} C_VEL
LIN {X 0,Y 167.896,Z 379.264,A -85,B 0,C 180,E1 -26127.417,E2 -26127.417} C_VEL
LIN {X 0,Y 171.192,Z 387.8,A -85,B 0,C 180,E1 -26130.193,E2 -26130.193} C_VEL
LIN {X 0,Y 171.402,Z 388.486,A -85,B 0,C 180,E1 -26130.37,E2 -26130.37} C_VEL
LIN {X 0,Y 167.74,Z 429.063,A -85,B 0,C 180,E1 -26131.669,E2 -26131.669} C_VEL
LIN {X 0,Y 165.181,Z 443.2,A -85,B 0,C 180,E1 -26132.405,E2 -26132.405} C_VEL
LIN {X 0,Y 161.651,Z 456.53,A -85,B 0,C 180,E1 -26133.468,E2 -26133.468} C_VEL
LIN {X 0,Y 157.439,Z 468.787,A -85,B 0,C 180,E1 -26134.891,E2 -26134.891} C_VEL
LIN {X 0,Y 152.289,Z 480.658,A -85,B 0,C 180,E1 -26136.752,E2 -26136.752} C_VEL
LIN {X 0,Y 146.775,Z 491.324,A -85,B 0,C 180,E1 -26138.989,E2 -26138.989} C_VEL
LIN {X 0,Y 140.841,Z 500.885,A -85,B 0,C 180,E1 -26141.54,E2 -26141.54} C_VEL
LIN {X 0,Y 134.099,Z 510.416,A -85,B 0,C 180,E1 -26144.967,E2 -26144.967} C_VEL
LIN {X 0,Y 127.905,Z 518.15,A -85,B 0,C 180,E1 -26148.749,E2 -26148.749} C_VEL
LIN {X 0,Y 122.273,Z 524.446,A -85,B 0,C 180,E1 -26152.878,E2 -26152.878} C_VEL
LIN {X 0,Y 117.496,Z 529.527,A -85,B 0,C 180,E1 -26157.43,E2 -26157.43} C_VEL
LIN {X 0,Y 113.391,Z 533.538,A -85,B 0,C 180,E1 -26162.3,E2 -26162.3} C_VEL
LIN {X 0,Y 109.983,Z 536.595,A -85,B 0,C 180,E1 -26167.455,E2 -26167.455} C_VEL
LIN {X 0,Y 106.998,Z 539.317,A -85,B 0,C 180,E1 -26174.768,E2 -26174.768} C_VEL
LIN {X 0,Y 105.456,Z 540.533,A -85,B 0,C 180,E1 -26182.34,E2 -26182.34} C_VEL
LIN {X 0,Y 105.225,Z 540.305,A -85,B 0,C 180,E1 -26190,E2 -26190} C_VEL
LIN {X 0,Y 105.503,Z 539.665,A -85,B 0,C 180,E1 -26193.819,E2 -26193.819} C_VEL
LIN {X 0,Y 106.982,Z 537.311,A -85,B 0,C 180,E1 -26201.366,E2 -26201.366} C_VEL
LIN {X 0,Y 109.049,Z 534.505,A -85,B 0,C 180,E1 -26206.858,E2 -26206.858} C_VEL
LIN {X 0,Y 111.924,Z 530.783,A -85,B 0,C 180,E1 -26212.132,E2 -26212.132} C_VEL
LIN {X 0,Y 115.68,Z 526.044,A -85,B 0,C 180,E1 -26217.106,E2 -26217.106} C_VEL
LIN {X 0,Y 121.075,Z 519.052,A -85,B 0,C 180,E1 -26222.474,E2 -26222.474} C_VEL
LIN {X 0,Y 126.315,Z 511.591,A -85,B 0,C 180,E1 -26226.734,E2 -26226.734} C_VEL
LIN {X 0,Y 132.294,Z 502.434,A -85,B 0,C 180,E1 -26230.598,E2 -26230.598} C_VEL
LIN {X 0,Y 137.676,Z 493.094,A -85,B 0,C 180,E1 -26233.561,E2 -26233.561} C_VEL
LIN {X 0,Y 142.671,Z 482.901,A -85,B 0,C 180,E1 -26236.089,E2 -26236.089} C_VEL
LIN {X 0,Y 147.286,Z 472.254,A -85,B 0,C 180,E1 -26238.043,E2 -26238.043} C_VEL
LIN {X 0,Y 151.736,Z 459.441,A -85,B 0,C 180,E1 -26239.837,E2 -26239.837} C_VEL
LIN {X 0,Y 155.072,Z 446.976,A -85,B 0,C 180,E1 -26241.107,E2 -26241.107} C_VEL
LIN {X 0,Y 157.619,Z 434.178,A -85,B 0,C 180,E1 -26241.975,E2 -26241.975} C_VEL
LIN {X 0,Y 159.257,Z 419.831,A -85,B 0,C 180,E1 -26242.591,E2 -26242.591} C_VEL
LIN {X 0,Y 162.442,Z 380.217,A -85,B 0,C 180,E1 -26243.941,E2 -26243.941} C_VEL
LIN {X 0,Y 159.235,Z 371.528,A -85,B 0,C 180,E1 -26246.428,E2 -26246.428} C_VEL
LIN {X 0,Y 155.209,Z 362.244,A -85,B 0,C 180,E1 -26249.844,E2 -26249.844} C_VEL
LIN {X 0,Y 151.337,Z 354.276,A -85,B 0,C 180,E1 -26253.65,E2 -26253.65} C_VEL
LIN {X 0,Y 148.626,Z 349.42,A -85,B 0,C 180,E1 -26256.744,E2 -26256.744} C_VEL
LIN {X 0,Y 146.03,Z 344.834,A -85,B 0,C 180,E1 -26260.311,E2 -26260.311} C_VEL
LIN {X 0,Y 142.964,Z 339.683,A -85,B 0,C 180,E1 -26265.986,E2 -26265.986} C_VEL
LIN {X 0,Y 140.789,Z 336.223,A -85,B 0,C 180,E1 -26273.478,E2 -26273.478} C_VEL
LIN {X 0,Y 140.581,Z 335.035,A -85,B 0,C 180,E1 -26278.932,E2 -26278.932} C_VEL
LIN {X 0,Y 140.828,Z 335.649,A -85,B 0,C 180,E1 -26281.786,E2 -26281.786} C_VEL
LIN {X 0,Y 143.09,Z 338.748,A -85,B 0,C 180,E1 -26289.474,E2 -26289.474} C_VEL
LIN {X 0,Y 146.59,Z 344.342,A -85,B 0,C 180,E1 -26295.734,E2 -26295.734} C_VEL
LIN {X 0,Y 149.444,Z 348.94,A -85,B 0,C 180,E1 -26299.431,E2 -26299.431} C_VEL
LIN {X 0,Y 152.397,Z 354.258,A -85,B 0,C 180,E1 -26302.656,E2 -26302.656} C_VEL
LIN {X 0,Y 155.533,Z 360.193,A -85,B 0,C 180,E1 -26305.62,E2 -26305.62} C_VEL
LIN {X 0,Y 159.627,Z 369.04,A -85,B 0,C 180,E1 -26309.056,E2 -26309.056} C_VEL
LIN {X 0,Y 162.879,Z 377.201,A -85,B 0,C 180,E1 -26311.544,E2 -26311.544} C_VEL
LIN {X 0,Y 158.292,Z 429.567,A -85,B 0,C 180,E1 -26313.384,E2 -26313.384} C_VEL
LIN {X 0,Y 156.046,Z 443.119,A -85,B 0,C 180,E1 -26314.163,E2 -26314.163} C_VEL
LIN {X 0,Y 152.76,Z 456.344,A -85,B 0,C 180,E1 -26315.254,E2 -26315.254} C_VEL
LIN {X 0,Y 149.028,Z 468.345,A -85,B 0,C 180,E1 -26316.709,E2 -26316.709} C_VEL
LIN {X 0,Y 144.052,Z 480.887,A -85,B 0,C 180,E1 -26318.685,E2 -26318.685} C_VEL
LIN {X 0,Y 138.985,Z 491.959,A -85,B 0,C 180,E1 -26321.098,E2 -26321.098} C_VEL
LIN {X 0,Y 133.801,Z 501.541,A -85,B 0,C 180,E1 -26323.762,E2 -26323.762} C_VEL
LIN {X 0,Y 128.513,Z 510.235,A -85,B 0,C 180,E1 -26326.877,E2 -26326.877} C_VEL
LIN {X 0,Y 122.776,Z 518.926,A -85,B 0,C 180,E1 -26330.975,E2 -26330.975} C_VEL
LIN {X 0,Y 117.739,Z 526.056,A -85,B 0,C 180,E1 -26335.455,E2 -26335.455} C_VEL
LIN {X 0,Y 113.551,Z 531.902,A -85,B 0,C 180,E1 -26340.322,E2 -26340.322} C_VEL
LIN {X 0,Y 110.199,Z 536.622,A -85,B 0,C 180,E1 -26345.51,E2 -26345.51} C_VEL
LIN {X 0,Y 107.554,Z 540.341,A -85,B 0,C 180,E1 -26350.931,E2 -26350.931} C_VEL
LIN {X 0,Y 105.589,Z 543.908,A -85,B 0,C 180,E1 -26358.482,E2 -26358.482} C_VEL
LIN {X 0,Y 105.151,Z 545.122,A -85,B 0,C 180,E1 -26362.318,E2 -26362.318} C_VEL
LIN {X 0,Y 105.018,Z 545.955,A -85,B 0,C 180,E1 -26366.163,E2 -26366.163} C_VEL
LIN {X 0,Y 105.165,Z 546.406,A -85,B 0,C 180,E1 -26370,E2 -26370} C_VEL
LIN {X 0,Y 105.031,Z 546.479,A -85,B 0,C 180,E1 -26373.837,E2 -26373.837} C_VEL
LIN {X 0,Y 105.633,Z 545.547,A -85,B 0,C 180,E1 -26381.513,E2 -26381.513} C_VEL
LIN {X 0,Y 107.648,Z 543.17,A -85,B 0,C 180,E1 -26389.052,E2 -26389.052} C_VEL
LIN {X 0,Y 110.361,Z 540.383,A -85,B 0,C 180,E1 -26394.452,E2 -26394.452} C_VEL
LIN {X 0,Y 113.812,Z 536.702,A -85,B 0,C 180,E1 -26399.604,E2 -26399.604} C_VEL
LIN {X 0,Y 118.057,Z 532.039,A -85,B 0,C 180,E1 -26404.439,E2 -26404.439} C_VEL
LIN {X 0,Y 124.082,Z 525.164,A -85,B 0,C 180,E1 -26409.583,E2 -26409.583} C_VEL
LIN {X 0,Y 129.031,Z 519.12,A -85,B 0,C 180,E1 -26412.991,E2 -26412.991} C_VEL
LIN {X 0,Y 131.233,Z 515.608,A -85,B 0,C 180,E1 -26414.836,E2 -26414.836} C_VEL
LIN {X 0,Y 133.602,Z 509.616,A -85,B 0,C 180,E1 -26418.115,E2 -26418.115} C_VEL
LIN {X 0,Y 136.14,Z 503.207,A -85,B 0,C 180,E1 -26421.14,E2 -26421.14} C_VEL
LIN {X 0,Y 138.497,Z 498.922,A -85,B 0,C 180,E1 -26422.545,E2 -26422.545} C_VEL
LIN {X 0,Y 144.767,Z 488.164,A -85,B 0,C 180,E1 -26425.007,E2 -26425.007} C_VEL
LIN {X 0,Y 150.737,Z 476.03,A -85,B 0,C 180,E1 -26427.058,E2 -26427.058} C_VEL
LIN {X 0,Y 155.499,Z 464.123,A -85,B 0,C 180,E1 -26428.547,E2 -26428.547} C_VEL
LIN {X 0,Y 159.694,Z 450.865,A -85,B 0,C 180,E1 -26429.731,E2 -26429.731} C_VEL
LIN {X 0,Y 162.838,Z 437.237,A -85,B 0,C 180,E1 -26430.571,E2 -26430.571} C_VEL
LIN {X 0,Y 164.827,Z 423.351,A -85,B 0,C 180,E1 -26431.134,E2 -26431.134} C_VEL
LIN {X 0,Y 168.075,Z 388.344,A -85,B 0,C 180,E1 -26432.23,E2 -26432.23} C_VEL
LIN {X 0,Y 164.661,Z 379.84,A -85,B 0,C 180,E1 -26435.409,E2 -26435.409} C_VEL
LIN {X 0,Y 161.537,Z 372.984,A -85,B 0,C 180,E1 -26438.716,E2 -26438.716} C_VEL
LIN {X 0,Y 158.706,Z 367.194,A -85,B 0,C 180,E1 -26442.288,E2 -26442.288} C_VEL
LIN {X 0,Y 156.102,Z 362.614,A -85,B 0,C 180,E1 -26446.329,E2 -26446.329} C_VEL
LIN {X 0,Y 153.918,Z 358.592,A -85,B 0,C 180,E1 -26451.177,E2 -26451.177} C_VEL
LIN {X 0,Y 152.753,Z 356.76,A -85,B 0,C 180,E1 -26455.383,E2 -26455.383} C_VEL
LIN {X 0,Y 152.32,Z 355.668,A -85,B 0,C 180,E1 -26460.001,E2 -26460.001} C_VEL
LIN {X 0,Y 152.912,Z 357.548,A -85,B 0,C 180,E1 -26466.268,E2 -26466.268} C_VEL
LIN {X 0,Y 154.532,Z 360.751,A -85,B 0,C 180,E1 -26471.312,E2 -26471.312} C_VEL
LIN {X 0,Y 157.1,Z 365.848,A -85,B 0,C 180,E1 -26476.237,E2 -26476.237} C_VEL
LIN {X 0,Y 159.465,Z 370.783,A -85,B 0,C 180,E1 -26479.647,E2 -26479.647} C_VEL
LIN {X 0,Y 162.166,Z 376.772,A -85,B 0,C 180,E1 -26482.874,E2 -26482.874} C_VEL
LIN {X 0,Y 165.641,Z 385.587,A -85,B 0,C 180,E1 -26486.457,E2 -26486.457} C_VEL
LIN {X 0,Y 167.701,Z 391.325,A -85,B 0,C 180,E1 -26488.362,E2 -26488.362} C_VEL
LIN {X 0,Y 164.152,Z 429.056,A -85,B 0,C 180,E1 -26489.556,E2 -26489.556} C_VEL
LIN {X 0,Y 161.676,Z 442.548,A -85,B 0,C 180,E1 -26490.238,E2 -26490.238} C_VEL
LIN {X 0,Y 158.191,Z 455.499,A -85,B 0,C 180,E1 -26491.217,E2 -26491.217} C_VEL
LIN {X 0,Y 154.159,Z 467.155,A -85,B 0,C 180,E1 -26492.5,E2 -26492.5} C_VEL
LIN {X 0,Y 148.858,Z 479.338,A -85,B 0,C 180,E1 -26494.291,E2 -26494.291} C_VEL
LIN {X 0,Y 143.356,Z 489.817,A -85,B 0,C 180,E1 -26496.381,E2 -26496.381} C_VEL
LIN {X 0,Y 137.493,Z 499.224,A -85,B 0,C 180,E1 -26498.785,E2 -26498.785} C_VEL
LIN {X 0,Y 130.285,Z 509.061,A -85,B 0,C 180,E1 -26502.123,E2 -26502.123} C_VEL
LIN {X 0,Y 123.67,Z 517.07,A -85,B 0,C 180,E1 -26505.882,E2 -26505.882} C_VEL
LIN {X 0,Y 116.678,Z 524.587,A -85,B 0,C 180,E1 -26510.769,E2 -26510.769} C_VEL
LIN {X 0,Y 111.545,Z 529.677,A -85,B 0,C 180,E1 -26515.455,E2 -26515.455} C_VEL
LIN {X 0,Y 107.132,Z 533.698,A -85,B 0,C 180,E1 -26520.528,E2 -26520.528} C_VEL
LIN {X 0,Y 103.432,Z 536.765,A -85,B 0,C 180,E1 -26525.941,E2 -26525.941} C_VEL
LIN {X 0,Y 100.141,Z 539.498,A -85,B 0,C 180,E1 -26533.697,E2 -26533.697} C_VEL
LIN {X 0,Y 99.091,Z 540.306,A -85,B 0,C 180,E1 -26537.715,E2 -26537.715} C_VEL
LIN {X 0,Y 98.109,Z 540.797,A -85,B 0,C 180,E1 -26545.892,E2 -26545.892} C_VEL
LIN {X 0,Y 98.145,Z 540.512,A -85,B 0,C 180,E1 -26550,E2 -26550} C_VEL
